WH_DATA.0	 := GVL1.hwo_digitalAlarms[6].0	;	(*	DI:97	WH ALARM MUTE P/B	*)
WH_DATA.1	 := GVL1.hwo_digitalAlarms[6].1	;	(*	DI:98	STGR JOYSTICK CONTROL FAIL ALARM	*)
WH_DATA.2	 := GVL1.hwo_digitalAlarms[6].2	;	(*	DI:99	GEN.ALARM MAIN SUPPLY FAILURE	*)
WH_DATA.3	 := GVL1.hwo_digitalAlarms[6].3	;	(*	DI:100	GEN.ALARM ALT.SUPPLY FAILURE	*)
WH_DATA.4	 := GVL1.hwo_digitalAlarms[6].4	;	(*	DI:101	NAV.LIGHT POWER FAILURE	*)
WH_DATA.5	 := GVL1.hwo_digitalAlarms[6].5	;	(*	DI:102	NAV.LIGHT SYSTEM FAULT	*)
WH_DATA.6	 := GVL1.hwo_digitalAlarms[6].6	;	(*	DI:103	FIRE ALARM SYSTEM FAULT	*)
WH_DATA.7	 := GVL1.hwo_digitalAlarms[6].7	;	(*	DI:104	FIRE ALARM ACTVATED	*)
WH_DATA.8	 := GVL1.hwo_digitalAlarms[6].8	;	(*	DI:105	AUTO PILOT FAIL ALARM	*)
WH_DATA.9	 := GVL1.hwo_digitalAlarms[6].9	;	(*	DI:106	GAS DETECTION SYSTEM POWER FAIL	*)
WH_DATA.10	 := GVL1.hwo_digitalAlarms[6].10	;	(*	DI:107	H2S ALARM ACTIVATED	*)
WH_DATA.11	 := GVL1.hwo_digitalAlarms[6].11	;	(*	DI:108	LEL ALARM ACTIVATED	*)
WH_DATA.12	 := GVL1.hwo_digitalAlarms[6].12	;	(*	DI:109	WH AREA REF. LEAKAGE ALARM 	*)
WH_DATA.13	 := GVL1.hwo_digitalAlarms[6].13	;	(*	DI:110	PASSENGER AREA REF. LEAKAGE ALARM 	*)
WH_DATA.14	 := GVL1.hwo_digitalAlarms[6].14	;	(*	DI:111	DEPTH BELOW KEEL LOWER THAN SET.P 	*)
WH_DATA.15	 := GVL1.hwo_digitalAlarms[6].15	;	(*	DI:112	GMDSS COMMON ALRM	*)
						
MP1_DATA.0	 := GVL1.hwo_digitalAlarms[7].0	;	(*	DI:113	PORT ME COMMON ALARM	*)
MP1_DATA.1	 := GVL1.hwo_digitalAlarms[7].1	;	(*	DI:114	STBD ME COMMON ALARM	*)
MP1_DATA.2	 := GVL1.hwo_digitalAlarms[7].2	;	(*	DI:115	CENTER ME COMMON ALARM	*)
MP1_DATA.3	 := GVL1.hwo_digitalEvents[7].3	;	(*	DI:116	AUX COOLING PUMP-1 RUNNING	*)
MP1_DATA.4	 := GVL1.hwo_digitalAlarms[7].4	;	(*	DI:117	AUX COOLING PUMP-1 TRIP	*)
MP1_DATA.5	 := GVL1.hwo_digitalAlarms[7].5	;	(*	DI:118	FO PURIFIER COMMON ALRM	*)
MP1_DATA.6	 := GVL1.hwo_digitalAlarms[7].6	;	(*	DI:119	MSB: PREF. TRIP ALARM	*)
MP1_DATA.7	 := GVL1.hwo_digitalAlarms[7].7	;	(*	DI:120	MSB: 440V EARTH FAULT ALARM	*)
MP1_DATA.8	 := GVL1.hwo_digitalAlarms[7].8	;	(*	DI:121	MSB: 220V EARTH FAULT ALARM	*)
MP1_DATA.9	 := GVL1.hwo_digitalAlarms[7].9	;	(*	DI:122	MSB: 24VDC SUPPLY FAIL ALARM	*)
MP1_DATA.10	 := GVL1.hwo_digitalAlarms[7].10	;	(*	DI:123	MSB: ABNORMAL ALARM	*)
MP1_DATA.11	 := GVL1.hwo_digitalAlarms[7].11	;	(*	DI:124	AMS AC SUPPLY FAIL	*)
MP1_DATA.12	 := GVL1.hwo_digitalAlarms[7].12	;	(*	DI:125	AMS DC SUPPLY FAIL	*)
MP1_DATA.13	 := GVL1.hwo_digitalAlarms[7].13	;	(*	DI:126	ALRM MUTE AMS PANEL	*)
MP1_DATA.14	 := GVL1.hwo_digitalAlarms[7].14	;	(*	DI:127	BT ENGINE COMMON ALARM	*)
MP1_DATA.15	 := GVL1.hwo_digitalAlarms[7].15	;	(*	DI:128	ACCOM PASSAGE REF. LEAKAGE ALARM	*)
						
MP2_DATA.0	 := GVL1.hwo_digitalAlarms[8].0	;	(*	DI:129	SPARE	*)
MP2_DATA.1	 := GVL1.hwo_digitalAlarms[8].1	;	(*	DI:130	SPARE	*)
MP2_DATA.2	 := GVL1.hwo_digitalAlarms[8].2	;	(*	DI:131	SPARE	*)
MP2_DATA.3	 := GVL1.hwo_digitalAlarms[8].3	;	(*	DI:132	SPARE	*)
MP2_DATA.4	 := GVL1.hwo_digitalAlarms[8].4	;	(*	DI:133	SPARE	*)
MP2_DATA.5	 := GVL1.hwo_digitalAlarms[8].5	;	(*	DI:134	SPARE	*)
MP2_DATA.6	 := GVL1.hwo_digitalAlarms[8].6	;	(*	DI:135	SPARE	*)
MP2_DATA.7	 := GVL1.hwo_digitalAlarms[8].7	;	(*	DI:136	SPARE	*)
MP2_DATA.8	 := GVL1.hwo_digitalAlarms[8].8	;	(*	DI:137	SPARE	*)
MP2_DATA.9	 := GVL1.hwo_digitalAlarms[8].9	;	(*	DI:138	SPARE	*)
MP2_DATA.10	 := GVL1.hwo_digitalAlarms[8].10	;	(*	DI:139	SPARE	*)
MP2_DATA.11	 := GVL1.hwo_digitalAlarms[8].11	;	(*	DI:140	SPARE	*)
MP2_DATA.12	 := GVL1.hwo_digitalAlarms[8].12	;	(*	DI:141	SPARE	*)
MP2_DATA.13	 := GVL1.hwo_digitalAlarms[8].13	;	(*	DI:142	SPARE	*)
MP2_DATA.14	 := GVL1.hwo_digitalAlarms[8].14	;	(*	DI:143	SPARE	*)
MP2_DATA.15	 := GVL1.hwo_digitalAlarms[8].15	;	(*	DI:144	SPARE	*)
						
MP3_DATA.0	 := GVL1.hwo_digitalAlarms[9].0	;	(*	DI:145	SPARE	*)
MP3_DATA.1	 := GVL1.hwo_digitalAlarms[9].1	;	(*	DI:146	SPARE	*)
MP3_DATA.2	 := GVL1.hwo_digitalAlarms[9].2	;	(*	DI:147	SPARE	*)
MP3_DATA.3	 := GVL1.hwo_digitalAlarms[9].3	;	(*	DI:148	SPARE	*)
MP3_DATA.4	 := GVL1.hwo_digitalAlarms[9].4	;	(*	DI:149	SPARE	*)
MP3_DATA.5	 := GVL1.hwo_digitalAlarms[9].5	;	(*	DI:150	SPARE	*)
MP3_DATA.6	 := GVL1.hwo_digitalAlarms[9].6	;	(*	DI:151	SPARE	*)
MP3_DATA.7	 := GVL1.hwo_digitalAlarms[9].7	;	(*	DI:152	SPARE	*)
						
IF NOT GVL1.hwo_digitalAlarms[12].11 THEN						
AI1_DATA	:= REAL_TO_WORD (GVL1.hro_Ch0OutVal[2])	;	(*	AI:01-FRESH WATER TANK 1C	*)
AI2_DATA	:= REAL_TO_WORD (GVL1.hro_Ch1OutVal[2])	;	(*	AI:02-FRESH WATER TANK 2C	*)
AI3_DATA	:= REAL_TO_WORD (GVL1.hro_Ch2OutVal[2])	;	(*	AI:03-BLACK WATER TANK	*)
AI4_DATA	:= REAL_TO_WORD (GVL1.hro_Ch3OutVal[2])	;	(*	AI:04-GREY WATER TANK 	*)
AI5_DATA	:= REAL_TO_WORD (GVL1.hro_Ch4OutVal[2])	;	(*	AI:05-FUEL OIL TANK PORT 1P	*)
AI6_DATA	:= REAL_TO_WORD (GVL1.hro_Ch5OutVal[2])	;	(*	AI:06-FUEL OIL TANK STBD 1S	*)
AI7_DATA	:= REAL_TO_WORD (GVL1.hro_Ch6OutVal[2])	;	(*	AI:07-FUEL OIL TANK PORT 3C	*)
AI8_DATA	:= REAL_TO_WORD (GVL1.hro_Ch7OutVal[2])	;	(*	AI:08-BILGE HOLDING TANK	*)
AI9_DATA	:= REAL_TO_WORD (GVL1.hro_Ch8OutVal[2])	;	(*	AI:09-FODS TANK PORT	*)
AI10_DATA	:= REAL_TO_WORD (GVL1.hro_Ch9OutVal[2])	;	(*	AI:10-FODS TANK STDB	*)
AI11_DATA	:= REAL_TO_WORD (GVL1.hro_Ch10OutVal[2])	;	(*	AI:11-SLOPE TANK 	*)
AI12_DATA	:= REAL_TO_WORD (GVL1.hro_Ch11OutVal[2])	;	(*	AI:12-FUEL OIL TANK PORT 2C	*)
AI13_DATA	:= REAL_TO_WORD (GVL1.hro_Ch12OutVal[2])	;	(*	AI:13-FUEL OIL TANK PORT 4P	*)
AI14_DATA	:= REAL_TO_WORD (GVL1.hro_Ch13OutVal[2])	;	(*	AI:14-FUEL OIL TANK STBD 4S	*)

						
						
ELSE						
AI1_DATA	:= 0 ;					
AI2_DATA	:= 0 ;					
AI3_DATA	:= 0 ;					
AI4_DATA	:= 0 ;					
AI5_DATA	:= 0 ;					
AI6_DATA	:= 0 ;					
AI7_DATA	:= 0 ;					
AI8_DATA	:= 0 ;					
AI9_DATA	:= 0 ;					
AI10_DATA	:= 0 ;					
AI11_DATA	:= 0 ;					
AI12_DATA	:= 0 ;					
AI13_DATA	:= 0 ;					
AI14_DATA	:= 0 ;					
END_IF						
						
COM_DATA.0	 := GVL1.hwo_digitalAlarms[12].0	;(*	JB1 DI MODULE COMMS: FAIL	*)		
COM_DATA.1	 := GVL1.hwo_digitalAlarms[12].1	;(*	JB2 DI MODULE COMMS: FAIL	*)		
COM_DATA.2	 := GVL1.hwo_digitalAlarms[12].2	;(*	JB3 DI MODULE COMMS: FAIL	*)		
COM_DATA.3	 := GVL1.hwo_digitalAlarms[12].3	;(*	JB4 DI MODULE COMMS: FAIL	*)		
COM_DATA.4	 := GVL1.hwo_digitalAlarms[12].4	;(*	JB5 DI MODULE COMMS: FAIL	*)		
COM_DATA.5	 := GVL1.hwo_digitalAlarms[12].5	;(*	JB6 DI MODULE COMMS: FAIL	*)		
COM_DATA.6	 := GVL1.hwo_digitalAlarms[12].6	;(*	WH DI MODULE COMMS: FAIL	*)		
COM_DATA.7	 := GVL1.hwo_digitalAlarms[12].7	;(*	MP DI1 MODULE COMMS: FAIL	*)		
COM_DATA.8	 := GVL1.hwo_digitalAlarms[12].8	;(*	MP DI2 MODULE COMMS: FAIL	*)		
COM_DATA.9	 := GVL1.hwo_digitalAlarms[12].9	;(*	MP DIO MODULE COMMS: FAIL	*)		
COM_DATA.10	 := GVL1.hwo_digitalAlarms[12].10	;(*	MP DO MODULE COMMS: FAIL	*)		
COM_DATA.11	 := GVL1.hwo_digitalAlarms[12].11	;(*	MP AI MODULE COMMS: FAIL	*)		
COM_DATA.12	 := GVL1.hwo_digitalAlarms[12].12	; (*	ECR HMI COMMS: FAIL	*)		
COM_DATA.13	 := GVL1.hwo_digitalAlarms[12].13	; (*	WH HMI COMMS: FAIL	*)		
COM_DATA.14	 := GVL1.hwo_digitalAlarms[12].14	; (*	MESS HMI COMMS: FAIL	*)	
	
TK_AL1.0	:=	 GVL1.hwo_analogAlm[0].0   	OR	GVL1.hwo_analogAlm[0].1 	;	(*	AI:01-FW 1C LOW	*)
TK_AL1.1	:=	 GVL1.hwo_analogAlm[0].2	OR	GVL1.hwo_analogAlm[0].5	;	(*	AI:01-FW 1C HIGH	*)
TK_AL1.2	:=	 GVL1.hwo_analogAlm[0].3	OR	GVL1.hwo_analogAlm[0].4	;	(*	AI:01-FW 1C FAULT	*)
TK_AL1.3	:=	 GVL1.hwo_analogAlm[1].0   	OR	GVL1.hwo_analogAlm[1].1 	;	(*	AI:02-FW 2C LOW	*)
TK_AL1.4	:=	 GVL1.hwo_analogAlm[1].2	OR	GVL1.hwo_analogAlm[1].5	;	(*	AI:02-FW 2C HIGH	*)
TK_AL1.5	:=	 GVL1.hwo_analogAlm[1].3	OR	GVL1.hwo_analogAlm[1].4	;	(*	AI:02-FW 2C FAULT	*)
TK_AL1.6	:=	 GVL1.hwo_analogAlm[2].0   	OR	GVL1.hwo_analogAlm[2].1 	;	(*	AI:03-BW LOW	*)
TK_AL1.7	:=	 GVL1.hwo_analogAlm[2].2	OR	GVL1.hwo_analogAlm[2].5	;	(*	AI:03-BW HIGH	*)
TK_AL1.8	:=	 GVL1.hwo_analogAlm[2].3	OR	GVL1.hwo_analogAlm[2].4	;	(*	AI:03-BW FAULT	*)
TK_AL1.9	:=	 GVL1.hwo_analogAlm[3].0   	OR	GVL1.hwo_analogAlm[3].1 	;	(*	AI:04-GW LOW	*)
TK_AL1.10	:=	 GVL1.hwo_analogAlm[3].2	OR	GVL1.hwo_analogAlm[3].5	;	(*	AI:04-GW HIGH	*)
TK_AL1.11	:=	 GVL1.hwo_analogAlm[3].3	OR	GVL1.hwo_analogAlm[3].4	;	(*	AI:04-GW FAULT	*)
TK_AL1.12	:=	 GVL1.hwo_analogAlm[4].0   	OR	GVL1.hwo_analogAlm[4].1 	;	(*	AI:05-FOT1P LOW	*)
TK_AL1.13	:=	 GVL1.hwo_analogAlm[4].2	OR	GVL1.hwo_analogAlm[4].5	;	(*	AI:05-FOT1P HIGH	*)
TK_AL1.14	:=	 GVL1.hwo_analogAlm[4].3	OR	GVL1.hwo_analogAlm[4].4	;	(*	AI:05-FOT1P FAULT	*)
TK_AL1.15	:=	 GVL1.hwo_analogAlm[5].0   	OR	GVL1.hwo_analogAlm[5].1 	;	(*	AI:06-FOT1S LOW	*)
								
TK_AL2.0	:=	 GVL1.hwo_analogAlm[5].2	OR	GVL1.hwo_analogAlm[5].5	;	(*	AI:06-FOT1S HIGH	*)
TK_AL2.1	:=	 GVL1.hwo_analogAlm[5].3	OR	GVL1.hwo_analogAlm[5].4	;	(*	AI:06-FOT1S FAULT	*)
TK_AL2.2	:=	 GVL1.hwo_analogAlm[6].0   	OR	GVL1.hwo_analogAlm[6].1 	;	(*	AI:07-FOT3C LOW	*)
TK_AL2.3	:=	 GVL1.hwo_analogAlm[6].2	OR	GVL1.hwo_analogAlm[6].5	;	(*	AI:07-FOT3C HIGH	*)
TK_AL2.4	:=	 GVL1.hwo_analogAlm[6].3	OR	GVL1.hwo_analogAlm[6].4	;	(*	AI:07-FOT3C FAULT	*)
TK_AL2.5	:=	 GVL1.hwo_analogAlm[7].0   	OR	GVL1.hwo_analogAlm[7].1 	;	(*	AI:08-BILGE.H LOW	*)
TK_AL2.6	:=	 GVL1.hwo_analogAlm[7].2	OR	GVL1.hwo_analogAlm[7].5	;	(*	AI:08-BILGE.H HIGH	*)
TK_AL2.7	:=	 GVL1.hwo_analogAlm[7].3	OR	GVL1.hwo_analogAlm[7].4	;	(*	AI:08-BILGE.H FAULT	*)
TK_AL2.8	:=	 GVL1.hwo_analogAlm[8].0   	OR	GVL1.hwo_analogAlm[8].1 	;	(*	AI:09-FODS P LOW	*)
TK_AL2.9	:=	 GVL1.hwo_analogAlm[8].2	OR	GVL1.hwo_analogAlm[8].5	;	(*	AI:09-FODS P HIGH	*)
TK_AL2.10	:=	 GVL1.hwo_analogAlm[8].3	OR	GVL1.hwo_analogAlm[8].4	;	(*	AI:09-FODS P FAULT	*)
TK_AL2.11	:=	 GVL1.hwo_analogAlm[9].0   	OR	GVL1.hwo_analogAlm[9].1 	;	(*	AI:10-FODS S LOW	*)
TK_AL2.12	:=	 GVL1.hwo_analogAlm[9].2	OR	GVL1.hwo_analogAlm[9].5	;	(*	AI:10-FODS S HIGH	*)
TK_AL2.13	:=	 GVL1.hwo_analogAlm[9].3	OR	GVL1.hwo_analogAlm[9].4	;	(*	AI:10-FODS S FAULT	*)
TK_AL2.14	:=	 GVL1.hwo_analogAlm[10].0  	OR	GVL1.hwo_analogAlm[10].1 	;	(*	AI:11-SLOPE LOW	*)
TK_AL2.15	:=	 GVL1.hwo_analogAlm[10].2	OR	GVL1.hwo_analogAlm[10].5 	;	(*	AI:11-SLOPE HIGH	*)
								
TK_AL3.0	:=	 GVL1.hwo_analogAlm[10].3	OR	GVL1.hwo_analogAlm[10].4	;	(*	AI:11-SLOPE FAULT	*)
TK_AL3.1	:=	 GVL1.hwo_analogAlm[11].0  	OR	GVL1.hwo_analogAlm[11].1 	;	(*	AI:12-FOT2C LOW	*)
TK_AL3.2	:=	 GVL1.hwo_analogAlm[11].2	OR	GVL1.hwo_analogAlm[11].5	;	(*	AI:12-FOT2C HIGH	*)
TK_AL3.3	:=	 GVL1.hwo_analogAlm[11].3	OR	GVL1.hwo_analogAlm[11].4	;	(*	AI:12-FOT2C FAULT	*)
TK_AL3.4	:=	 GVL1.hwo_analogAlm[12].0 	OR	GVL1.hwo_analogAlm[12].1 	;	(*	AI:13-FOT4P LOW	*)
TK_AL3.5	:=	 GVL1.hwo_analogAlm[12].2	OR	GVL1.hwo_analogAlm[12].5	;	(*	AI:13-FOT4P HIGH	*)
TK_AL3.6	:=	 GVL1.hwo_analogAlm[12].3	OR	GVL1.hwo_analogAlm[12].4	;	(*	AI:13-FOT4P FAULT	*)
TK_AL3.7	:=	 GVL1.hwo_analogAlm[13].0 	OR	GVL1.hwo_analogAlm[13].1 	;	(*	AI:14-FOT4S LOW	*)
TK_AL3.8	:=	 GVL1.hwo_analogAlm[13].2	OR	GVL1.hwo_analogAlm[13].5	;	(*	AI:14-FOT4S HIGH	*)
TK_AL3.9	:=	 GVL1.hwo_analogAlm[13].3	OR	GVL1.hwo_analogAlm[13].4	;	(*	AI:14-FOT4S FAULT	*)
END_ACTION

END_PROGRAM

// Device/Application/fb_alarmEvent
FUNCTION_BLOCK fb_alarmEvent
VAR_INPUT
	wi_input: WORD;
	wi_set: WORD :=65535;
	wai_delay: ARRAY[0..15] OF WORD;
	wi_inhibit: WORD;
	wi_inhibitJm: WORD;
	wi_interlock: WORD;
	wi_alarmEvent: WORD;
	xi_reset: BOOL;
	xi_ack: BOOL;
	
END_VAR
VAR_OUTPUT
	wo_alarm: WORD;
	wo_event: WORD;
	wo_alarmLa : WORD;
	xo_buzzer: BOOL;
	xo_ind: BOOL;
	xo_indLa: BOOL;
	wo_inhTot: WORD;
END_VAR
VAR
	AlarmOutTemp: WORD;
	AlarmDelayTemp: ARRAY[0..15] OF TIME;
	

	HighInterlock1: WORD;
	HighInterlock2: WORD;
	LowInterlock1: WORD;
	LowInterlock2: WORD;
	
	TR1: TON;
	TR2: TON;
	TR3: TON;
	TR4: TON;
	TR5: TON;
	TR6: TON;
	TR7: TON;
	TR8: TON;
	TR9: TON;
	TR10: TON;
	TR11: TON;
	TR12: TON;
	TR13: TON;
	TR14: TON;
	TR15: TON;
	TR16: TON;
	AlarmOut1: TP;
	AlarmOut2: TP;
	AlarmOut3: TP;
	AlarmOut4: TP;
	AlarmOut5: TP;
	AlarmOut6: TP;
	AlarmOut7: TP;
	AlarmOut8: TP;
	AlarmOut9: TP;
	AlarmOut10: TP;
	AlarmOut11: TP;
	AlarmOut12: TP;
	AlarmOut13: TP;
	AlarmOut14: TP;
	AlarmOut15: TP;
	AlarmOut16: TP;
	x_reset1: BOOL;
	x_reset2: BOOL;
	x_reset3: BOOL;
	x_reset4: BOOL;
	x_reset5: BOOL;
	x_reset6: BOOL;
	x_reset7: BOOL;
	x_reset8: BOOL;
	x_reset9: BOOL;
	x_reset10: BOOL;
	x_reset11: BOOL;
	x_reset12: BOOL;
	x_reset13: BOOL;
	x_reset14: BOOL;
	x_reset15: BOOL;
	x_reset16: BOOL;
END_VAR

(*Alarm1*)

(*x_reset*)
IF wo_alarm.0 AND xi_reset THEN
x_reset1:= TRUE;
ELSE
x_reset1:= FALSE;
END_IF


(*Time delay*)
TR1(IN:= , PT:= , Q=> , ET=> );
TR1.IN:=AlarmOutTemp.0;
TR1.PT:= AlarmDelayTemp[0];
AlarmDelayTemp[0]:=WORD_TO_TIME ( wai_delay[0]*1000);

(*Alarm condition:- Set NO/NC, Inhibit, x_reset*)
IF ((wi_input.0=1 AND wi_set.0=1) OR (wi_input.0=0 AND wi_set.0=0)) AND wi_inhibit.0=0 AND wi_inhibitJm.0=0 AND x_reset1=0
THEN
AlarmOutTemp.0:=1;
ELSE
AlarmOutTemp.0:=0;
END_IF


(*Final alarm and event output with delay*)
wo_alarm.0:=TR1.Q AND wi_alarmEvent.0 AND NOT wi_interlock.0;
wo_event.0:=TR1.Q ;
(*Final alarm single pulse latched till acknowledge*)
AlarmOut1(IN:=wo_alarm.0 , PT:= T#1s, Q=> , ET=> );
IF (AlarmOut1.Q OR wo_alarmLa.0) AND NOT xi_ack THEN wo_alarmLa.0:=1; ELSE wo_alarmLa.0:=0; END_IF
(*------------------------------------------------------------------------------------------------------------------------------*)

(*Alarm2*)

(*x_reset*)
IF wo_alarm.1 AND xi_reset THEN
x_reset2:= TRUE;
ELSE
x_reset2:= FALSE;
END_IF


(*Time delay*)
TR2(IN:= , PT:= , Q=> , ET=> );
TR2.IN:=AlarmOutTemp.1;
TR2.PT:= AlarmDelayTemp[1];
AlarmDelayTemp[1]:=WORD_TO_TIME ( wai_delay[1]*1000);

(*Alarm condition:- Set NO/NC, Inhibit, x_reset*)
IF ((wi_input.1=1 AND wi_set.1=1) OR (wi_input.1=0 AND wi_set.1=0)) AND wi_inhibit.1=0 AND wi_inhibitJm.1=0  AND x_reset2=0
THEN
AlarmOutTemp.1:=1;
ELSE
AlarmOutTemp.1:=0;
END_IF


(*Final alarm and event output with delay*)
wo_alarm.1:=TR2.Q AND wi_alarmEvent.1 AND NOT wi_interlock.1;
wo_event.1:=TR2.Q;
(*Final alarm single pulse latched till acknowledge*)
AlarmOut2(IN:=wo_alarm.1 , PT:= T#1s, Q=> , ET=> );
IF (AlarmOut2.Q OR wo_alarmLa.1) AND NOT xi_ack THEN wo_alarmLa.1:=1; ELSE wo_alarmLa.1:=0; END_IF

(*------------------------------------------------------------------------------------------------------------------------------*)

(*Alarm3*)

(*x_reset*)
IF wo_alarm.2 AND xi_reset THEN
x_reset3:= TRUE;
ELSE
x_reset3:= FALSE;
END_IF


(*Time delay*)
TR3(IN:= , PT:= , Q=> , ET=> );
TR3.IN:=AlarmOutTemp.2;
TR3.PT:= AlarmDelayTemp[2];
AlarmDelayTemp[2]:=WORD_TO_TIME ( wai_delay[2]*1000);

(*Alarm condition:- Set NO/NC, Inhibit, x_reset*)
IF ((wi_input.2=1 AND wi_set.2=1) OR (wi_input.2=0 AND wi_set.2=0)) AND wi_inhibit.2=0 AND wi_inhibitJm.2=0   AND x_reset3=0
THEN
AlarmOutTemp.2:=1;
ELSE
AlarmOutTemp.2:=0;
END_IF

(*Final alarm and event output with delay*)
wo_alarm.2:=TR3.Q AND wi_alarmEvent.2 AND NOT wi_interlock.2;
wo_event.2:=TR3.Q;
(*Final alarm single pulse latched till acknowledge*)
AlarmOut3(IN:=wo_alarm.2 , PT:= T#1s, Q=> , ET=> );
IF (AlarmOut3.Q OR wo_alarmLa.2) AND NOT xi_ack THEN wo_alarmLa.2:=1; ELSE wo_alarmLa.2:=0; END_IF
(*------------------------------------------------------------------------------------------------------------------------------*)

(*Alarm4*)

(*x_reset*)
IF wo_alarm.3 AND xi_reset THEN
x_reset4:= TRUE;
ELSE
x_reset4:= FALSE;
END_IF


(*Time delay*)
TR4(IN:= , PT:= , Q=> , ET=> );
TR4.IN:=AlarmOutTemp.3;
TR4.PT:= AlarmDelayTemp[3];
AlarmDelayTemp[3]:=WORD_TO_TIME ( wai_delay[3]*1000);

(*Alarm condition:- Set NO/NC, Inhibit, x_reset*)
IF ((wi_input.3=1 AND wi_set.3=1) OR (wi_input.3=0 AND wi_set.3=0)) AND wi_inhibit.3=0 AND wi_inhibitJm.3=0  AND x_reset4=0
THEN
AlarmOutTemp.3:=1;
ELSE
AlarmOutTemp.3:=0;
END_IF

(*Final alarm and event output with delay*)
wo_alarm.3:=TR4.Q AND wi_alarmEvent.3 AND NOT wi_interlock.3;
wo_event.3:=TR4.Q;
(*Final alarm single pulse latched till acknowledge*)
AlarmOut4(IN:=wo_alarm.3 , PT:= T#1s, Q=> , ET=> );
IF (AlarmOut4.Q OR wo_alarmLa.3) AND NOT xi_ack THEN wo_alarmLa.3:=1; ELSE wo_alarmLa.3:=0; END_IF
(*------------------------------------------------------------------------------------------------------------------------------*)

(*Alarm5*)

(*x_reset*)
IF wo_alarm.4 AND xi_reset THEN
x_reset5:= TRUE;
ELSE
x_reset5:= FALSE;
END_IF


(*Time delay*)
TR5(IN:= , PT:= , Q=> , ET=> );
TR5.IN:=AlarmOutTemp.4;
TR5.PT:= AlarmDelayTemp[4];
AlarmDelayTemp[4]:=WORD_TO_TIME ( wai_delay[4]*1000);

(*Alarm condition:- Set NO/NC, Inhibit, x_reset*)
IF ((wi_input.4=1 AND wi_set.4=1) OR (wi_input.4=0 AND wi_set.4=0)) AND wi_inhibit.4=0 AND wi_inhibitJm.4=0   AND x_reset5=0
THEN
AlarmOutTemp.4:=1;
ELSE
AlarmOutTemp.4:=0;
END_IF

(*Final alarm and event output with delay*)
wo_alarm.4:=TR5.Q AND wi_alarmEvent.4 AND NOT wi_interlock.4;
wo_event.4:=TR5.Q;
(*Final alarm single pulse latched till acknowledge*)
AlarmOut5(IN:=wo_alarm.4 , PT:= T#1s, Q=> , ET=> );
IF (AlarmOut5.Q OR wo_alarmLa.4) AND NOT xi_ack THEN wo_alarmLa.4:=1; ELSE wo_alarmLa.4:=0; END_IF

(*------------------------------------------------------------------------------------------------------------------------------*)

(*Alarm6*)

(*x_reset*)
IF wo_alarm.5 AND xi_reset THEN
x_reset6:= TRUE;
ELSE
x_reset6:= FALSE;
END_IF


(*Time delay*)
TR6(IN:= , PT:= , Q=> , ET=> );
TR6.IN:=AlarmOutTemp.5;
TR6.PT:= AlarmDelayTemp[5];
AlarmDelayTemp[5]:=WORD_TO_TIME ( wai_delay[5]*1000);

(*Alarm condition:- Set NO/NC, Inhibit, x_reset*)
IF ((wi_input.5=1 AND wi_set.5=1) OR (wi_input.5=0 AND wi_set.5=0)) AND wi_inhibit.5=0 AND wi_inhibitJm.5=0   AND x_reset6=0
THEN
AlarmOutTemp.5:=1;
ELSE
AlarmOutTemp.5:=0;
END_IF

(*Final alarm and event output with delay*)
wo_alarm.5:=TR6.Q AND wi_alarmEvent.5 AND NOT wi_interlock.5;
wo_event.5:=TR6.Q;
(*Final alarm single pulse latched till acknowledge*)
AlarmOut6(IN:=wo_alarm.5 , PT:= T#1s, Q=> , ET=> );
IF (AlarmOut6.Q OR wo_alarmLa.5) AND NOT xi_ack THEN wo_alarmLa.5:=1; ELSE wo_alarmLa.5:=0; END_IF
(*------------------------------------------------------------------------------------------------------------------------------*)

(*Alarm7*)

(*x_reset*)
IF wo_alarm.6 AND xi_reset THEN
x_reset7:= TRUE;
ELSE
x_reset7:= FALSE;
END_IF


(*Time delay*)
TR7(IN:= , PT:= , Q=> , ET=> );
TR7.IN:=AlarmOutTemp.6;
TR7.PT:= AlarmDelayTemp[6];
AlarmDelayTemp[6]:=WORD_TO_TIME ( wai_delay[6]*1000);

(*Alarm condition:- Set NO/NC, Inhibit, x_reset*)
IF ((wi_input.6=1 AND wi_set.6=1) OR (wi_input.6=0 AND wi_set.6=0)) AND wi_inhibit.6=0 AND wi_inhibitJm.6=0   AND x_reset7=0
THEN
AlarmOutTemp.6:=1;
ELSE
AlarmOutTemp.6:=0;
END_IF


(*Final alarm and event output with delay*)
wo_alarm.6:=TR7.Q AND wi_alarmEvent.6 AND NOT wi_interlock.6;
wo_event.6:=TR7.Q;
(*Final alarm single pulse latched till acknowledge*)
AlarmOut7(IN:=wo_alarm.6 , PT:= T#1s, Q=> , ET=> );
IF (AlarmOut7.Q OR wo_alarmLa.6) AND NOT xi_ack THEN wo_alarmLa.6:=1; ELSE wo_alarmLa.6:=0; END_IF
(*------------------------------------------------------------------------------------------------------------------------------*)

(*Alarm8*)

(*x_reset*)
IF wo_alarm.7 AND xi_reset THEN
x_reset8:= TRUE;
ELSE
x_reset8:= FALSE;
END_IF


(*Time delay*)
TR8(IN:= , PT:= , Q=> , ET=> );
TR8.IN:=AlarmOutTemp.7;
TR8.PT:= AlarmDelayTemp[7];
AlarmDelayTemp[7]:=WORD_TO_TIME ( wai_delay[7]*1000);

(*Alarm condition:- Set NO/NC, Inhibit, x_reset*)
IF ((wi_input.7=1 AND wi_set.7=1) OR (wi_input.7=0 AND wi_set.7=0)) AND wi_inhibit.7=0 AND wi_inhibitJm.7=0   AND x_reset8=0
THEN
AlarmOutTemp.7:=1;
ELSE
AlarmOutTemp.7:=0;
END_IF

(*Final alarm and event output with delay*)
wo_alarm.7:=TR8.Q AND wi_alarmEvent.7 AND NOT wi_interlock.7;
wo_event.7:=TR8.Q;
(*Final alarm single pulse latched till acknowledge*)
AlarmOut8(IN:=wo_alarm.7 , PT:= T#1s, Q=> , ET=> );
IF (AlarmOut8.Q OR wo_alarmLa.7) AND NOT xi_ack THEN wo_alarmLa.7:=1; ELSE wo_alarmLa.7:=0; END_IF
(*------------------------------------------------------------------------------------------------------------------------------*)

(*Alarm9*)

(*x_reset*)
IF wo_alarm.8 AND xi_reset THEN
x_reset9:= TRUE;
ELSE
x_reset9:= FALSE;
END_IF


(*Time delay*)
TR9(IN:= , PT:= , Q=> , ET=> );
TR9.IN:=AlarmOutTemp.8;
TR9.PT:= AlarmDelayTemp[8];
AlarmDelayTemp[8]:=WORD_TO_TIME ( wai_delay[8]*1000);

(*Alarm condition:- Set NO/NC, Inhibit, x_reset*)
IF ((wi_input.8=1 AND wi_set.8=1) OR (wi_input.8=0 AND wi_set.8=0)) AND wi_inhibit.8=0 AND wi_inhibitJm.8=0   AND x_reset9=0
THEN
AlarmOutTemp.8:=1;
ELSE
AlarmOutTemp.8:=0;
END_IF

(*Final alarm and event output with delay*)
wo_alarm.8:=TR9.Q AND wi_alarmEvent.8 AND NOT wi_interlock.8;
wo_event.8:=TR9.Q;
(*Final alarm single pulse latched till acknowledge*)
AlarmOut9(IN:=wo_alarm.8 , PT:= T#1s, Q=> , ET=> );
IF (AlarmOut9.Q OR wo_alarmLa.8) AND NOT xi_ack THEN wo_alarmLa.8:=1; ELSE wo_alarmLa.8:=0; END_IF
(*------------------------------------------------------------------------------------------------------------------------------*)

(*Alarm10*)

(*x_reset*)
IF wo_alarm.9 AND xi_reset THEN
x_reset10:= TRUE;
ELSE
x_reset10:= FALSE;
END_IF


(*Time delay*)
TR10(IN:= , PT:= , Q=> , ET=> );
TR10.IN:=AlarmOutTemp.9;
TR10.PT:= AlarmDelayTemp[9];
AlarmDelayTemp[9]:=WORD_TO_TIME ( wai_delay[9]*1000);

(*Alarm condition:- Set NO/NC, Inhibit, x_reset*)
IF ((wi_input.9=1 AND wi_set.9=1) OR (wi_input.9=0 AND wi_set.9=0)) AND wi_inhibit.9=0 AND wi_inhibitJm.9=0  AND x_reset10=0
THEN
AlarmOutTemp.9:=1;
ELSE
AlarmOutTemp.9:=0;
END_IF

(*Final alarm and event output with delay*)
wo_alarm.9:=TR10.Q AND wi_alarmEvent.9 AND NOT wi_interlock.9;
wo_event.9:=TR10.Q;
(*Final alarm single pulse latched till acknowledge*)
AlarmOut10(IN:=wo_alarm.9 , PT:= T#1s, Q=> , ET=> );
IF (AlarmOut10.Q OR wo_alarmLa.9) AND NOT xi_ack THEN wo_alarmLa.9:=1; ELSE wo_alarmLa.9:=0; END_IF
(*------------------------------------------------------------------------------------------------------------------------------*)

(*Alarm11*)

(*x_reset*)
IF wo_alarm.10 AND xi_reset THEN
x_reset11:= TRUE;
ELSE
x_reset11:= FALSE;
END_IF


(*Time delay*)
TR11(IN:= , PT:= , Q=> , ET=> );
TR11.IN:=AlarmOutTemp.10;
TR11.PT:= AlarmDelayTemp[10];
AlarmDelayTemp[10]:=WORD_TO_TIME ( wai_delay[10]*1000);

(*Alarm condition:- Set NO/NC, Inhibit, x_reset*)
IF ((wi_input.10=1 AND wi_set.10=1) OR (wi_input.10=0 AND wi_set.10=0)) AND wi_inhibit.10=0 AND wi_inhibitJm.10=0   AND x_reset11=0
THEN
AlarmOutTemp.10:=1;
ELSE
AlarmOutTemp.10:=0;
END_IF

(*Final alarm and event output with delay*)
wo_alarm.10:=TR11.Q AND wi_alarmEvent.10 AND NOT wi_interlock.10;
wo_event.10:=TR11.Q;
(*Final alarm single pulse latched till acknowledge*)
AlarmOut11(IN:=wo_alarm.10 , PT:= T#1s, Q=> , ET=> );
IF (AlarmOut11.Q OR wo_alarmLa.10) AND NOT xi_ack THEN wo_alarmLa.10:=1; ELSE wo_alarmLa.10:=0; END_IF
(*------------------------------------------------------------------------------------------------------------------------------*)

(*Alarm12*)

(*x_reset*)
IF wo_alarm.11 AND xi_reset THEN
x_reset12:= TRUE;
ELSE
x_reset12:= FALSE;
END_IF


(*Time delay*)
TR12(IN:= , PT:= , Q=> , ET=> );
TR12.IN:=AlarmOutTemp.11;
TR12.PT:= AlarmDelayTemp[11];
AlarmDelayTemp[11]:=WORD_TO_TIME ( wai_delay[11]*1000);

(*Alarm condition:- Set NO/NC, Inhibit, x_reset*)
IF ((wi_input.11=1 AND wi_set.11=1) OR (wi_input.11=0 AND wi_set.11=0)) AND wi_inhibit.11=0 AND wi_inhibitJm.11=0   AND x_reset12=0
THEN
AlarmOutTemp.11:=1;
ELSE
AlarmOutTemp.11:=0;
END_IF

(*Final alarm and event output with delay*)
wo_alarm.11:=TR12.Q AND wi_alarmEvent.11 AND NOT wi_interlock.11;
wo_event.11:=TR12.Q;
(*Final alarm single pulse latched till acknowledge*)
AlarmOut12(IN:=wo_alarm.11 , PT:= T#1s, Q=> , ET=> );
IF (AlarmOut12.Q OR wo_alarmLa.11) AND NOT xi_ack THEN wo_alarmLa.11:=1; ELSE wo_alarmLa.11:=0; END_IF

(*------------------------------------------------------------------------------------------------------------------------------*)

(*Alarm13*)

(*x_reset*)
IF wo_alarm.12 AND xi_reset THEN
x_reset13:= TRUE;
ELSE
x_reset13:= FALSE;
END_IF


(*Time delay*)
TR13(IN:= , PT:= , Q=> , ET=> );
TR13.IN:=AlarmOutTemp.12;
TR13.PT:= AlarmDelayTemp[12];
AlarmDelayTemp[12]:=WORD_TO_TIME ( wai_delay[12]*1000);

(*Alarm condition:- Set NO/NC, Inhibit, x_reset*)
IF ((wi_input.12=1 AND wi_set.12=1) OR (wi_input.12=0 AND wi_set.12=0)) AND wi_inhibit.12=0 AND wi_inhibitJm.12=0   AND x_reset13=0
THEN
AlarmOutTemp.12:=1;
ELSE
AlarmOutTemp.12:=0;
END_IF

(*Final alarm and event output with delay*)
wo_alarm.12:=TR13.Q AND wi_alarmEvent.12 AND NOT wi_interlock.12;
wo_event.12:=TR13.Q;
(*Final alarm single pulse latched till acknowledge*)
AlarmOut13(IN:=wo_alarm.12 , PT:= T#1s, Q=> , ET=> );
IF (AlarmOut13.Q OR wo_alarmLa.12) AND NOT xi_ack THEN wo_alarmLa.12:=1; ELSE wo_alarmLa.12:=0; END_IF
(*------------------------------------------------------------------------------------------------------------------------------*)

(*Alarm14*)

(*x_reset*)
IF wo_alarm.13 AND xi_reset THEN
x_reset14:= TRUE;
ELSE
x_reset14:= FALSE;
END_IF


(*Time delay*)
TR14(IN:= , PT:= , Q=> , ET=> );
TR14.IN:=AlarmOutTemp.13;
TR14.PT:= AlarmDelayTemp[13];
AlarmDelayTemp[13]:=WORD_TO_TIME ( wai_delay[13]*1000);

(*Alarm condition:- Set NO/NC, Inhibit, x_reset*)
IF ((wi_input.13=1 AND wi_set.13=1) OR (wi_input.13=0 AND wi_set.13=0)) AND wi_inhibit.13=0 AND wi_inhibitJm.13=0   AND x_reset14=0
THEN
AlarmOutTemp.13:=1;
ELSE
AlarmOutTemp.13:=0;
END_IF

(*Final alarm and event output with delay*)
wo_alarm.13:=TR14.Q AND wi_alarmEvent.13 AND NOT wi_interlock.13;
wo_event.13:=TR14.Q;
(*Final alarm single pulse latched till acknowledge*)
AlarmOut14(IN:=wo_alarm.13 , PT:= T#1s, Q=> , ET=> );
IF (AlarmOut14.Q OR wo_alarmLa.13) AND NOT xi_ack THEN wo_alarmLa.13:=1; ELSE wo_alarmLa.13:=0; END_IF
(*------------------------------------------------------------------------------------------------------------------------------*)

(*Alarm15*)

(*x_reset*)
IF wo_alarm.14 AND xi_reset THEN
x_reset15:= TRUE;
ELSE
x_reset15:= FALSE;
END_IF


(*Time delay*)
TR15(IN:= , PT:= , Q=> , ET=> );
TR15.IN:=AlarmOutTemp.14;
TR15.PT:= AlarmDelayTemp[14];
AlarmDelayTemp[14]:=WORD_TO_TIME ( wai_delay[14]*1000);

(*Alarm condition:- Set NO/NC, Inhibit, x_reset*)
IF ((wi_input.14=1 AND wi_set.14=1) OR (wi_input.14=0 AND wi_set.14=0)) AND wi_inhibit.14=0 AND wi_inhibitJm.14=0  AND x_reset15=0
THEN
AlarmOutTemp.14:=1;
ELSE
AlarmOutTemp.14:=0;
END_IF


(*Final alarm and event output with delay*)
wo_alarm.14:=TR15.Q AND wi_alarmEvent.14 AND NOT wi_interlock.14;
wo_event.14:=TR15.Q;
(*Final alarm single pulse latched till acknowledge*)
AlarmOut15(IN:=wo_alarm.14 , PT:= T#1s, Q=> , ET=> );
IF(AlarmOut15.Q OR wo_alarmLa.14) AND NOT xi_ack THEN wo_alarmLa.14:=1; ELSE wo_alarmLa.14:=0; END_IF
(*------------------------------------------------------------------------------------------------------------------------------*)

(*Alarm16*)

(*x_reset*)
IF wo_alarm.15 AND xi_reset THEN
x_reset16:= TRUE;
ELSE
x_reset16:= FALSE;
END_IF


(*Time delay*)
TR16(IN:= , PT:= , Q=> , ET=> );
TR16.IN:=AlarmOutTemp.15;
TR16.PT:= AlarmDelayTemp[15];
AlarmDelayTemp[15]:=WORD_TO_TIME ( wai_delay[15]*1000);

(*Alarm condition:- Set NO/NC, Inhibit, x_reset*)
IF ((wi_input.15=1 AND wi_set.15=1) OR (wi_input.15=0 AND wi_set.15=0)) AND wi_inhibit.15=0 AND wi_inhibitJm.15=0  AND x_reset16=0
THEN
AlarmOutTemp.15:=1;
ELSE
AlarmOutTemp.15:=0;
END_IF


(*Final alarm and event output with delay*)
wo_alarm.15:=TR16.Q AND wi_alarmEvent.15 AND NOT wi_interlock.15;
wo_event.15:=TR16.Q;
(*Final alarm single pulse latched till acknowledge*)
AlarmOut16(IN:=wo_alarm.15 , PT:= T#1s, Q=> , ET=> );
IF (AlarmOut16.Q OR wo_alarmLa.15) AND NOT xi_ack THEN wo_alarmLa.15:=1; ELSE wo_alarmLa.15:=0; END_IF

(*common buzzer out*)

IF AlarmOut1.Q OR AlarmOut2.Q OR AlarmOut3.Q OR AlarmOut4.Q OR AlarmOut5.Q OR AlarmOut6.Q OR AlarmOut7.Q OR AlarmOut8.Q
OR AlarmOut9.Q OR AlarmOut10.Q OR AlarmOut11.Q OR AlarmOut12.Q OR AlarmOut13.Q OR AlarmOut14.Q OR AlarmOut15.Q OR AlarmOut16.Q THEN
xo_buzzer := 1;
ELSE
xo_buzzer := 0;
END_IF
(*common indication out*)
IF wo_alarm.0 OR wo_alarm.1 OR wo_alarm.2 OR wo_alarm.3 OR wo_alarm.4 OR wo_alarm.5 OR wo_alarm.6
OR wo_alarm.7 OR wo_alarm.8 OR wo_alarm.9 OR wo_alarm.10 OR wo_alarm.11 OR wo_alarm.12 OR wo_alarm.13
OR wo_alarm.14 OR wo_alarm.15 THEN
xo_ind := 1;
ELSE
xo_ind := 0;
END_IF
(*common indication out single pulse latched till acknowledge*)
IF wo_alarmLa.0 OR wo_alarmLa.1 OR wo_alarmLa.2 OR wo_alarmLa.3 OR wo_alarmLa.4 OR wo_alarmLa.5 OR wo_alarmLa.6
OR wo_alarmLa.7 OR wo_alarmLa.8 OR wo_alarmLa.9 OR wo_alarmLa.10 OR wo_alarmLa.11 OR wo_alarmLa.12 OR wo_alarmLa.13
OR wo_alarmLa.14 OR wo_alarmLa.15 THEN
xo_indLa := 1;
ELSE
xo_indLa := 0;
END_IF

(*Total inhibited alarms from Jmobile*)
wo_inhTot := BOOL_TO_WORD(wi_inhibitJm.0) + BOOL_TO_WORD(wi_inhibitJm.1) + BOOL_TO_WORD(wi_inhibitJm.2)
 + BOOL_TO_WORD(wi_inhibitJm.3) + BOOL_TO_WORD(wi_inhibitJm.4) + BOOL_TO_WORD(wi_inhibitJm.5) + BOOL_TO_WORD(wi_inhibitJm.6)
 + BOOL_TO_WORD(wi_inhibitJm.7) + BOOL_TO_WORD(wi_inhibitJm.8) + BOOL_TO_WORD(wi_inhibitJm.9) + BOOL_TO_WORD(wi_inhibitJm.10)
 + BOOL_TO_WORD(wi_inhibitJm.11) + BOOL_TO_WORD(wi_inhibitJm.12) + BOOL_TO_WORD(wi_inhibitJm.13) + BOOL_TO_WORD(wi_inhibitJm.14)
 + BOOL_TO_WORD(wi_inhibitJm.15);

END_FUNCTION_BLOCK

// Device/Application/fb_tankMonitor
FUNCTION_BLOCK fb_tankMonitor
VAR_INPUT
	wi_sensorVal	: WORD;
	wi_samplingIn	: ARRAY[0..20] OF  WORD;
	wi_samplingOut	: ARRAY[0..20] OF  WORD;

	wi_chPara	: WORD;(*0:inhL1, 1:inhL2, 2:inhL3, 3:inhCable break, 4:inhOver range, 5:buz en L1, 6:buz en L2, 7:buz en L3, 8:buz en err1, 9:buz en err2, 10:inhL4, 11:buz en L4, 12: Auto filter enable
							13:Fill input sensor min value and range when tank empty, 14: Fill input sensor max value and range when tank full*)
	wi_chParaJm	: WORD;	
	xi_comErr	:BOOL;
	xi_ack	:BOOL;
END_VAR
VAR_OUTPUT
	ro_pressOut	:REAL;
	ro_htOut	:REAL;
	ro_volOut	:REAL;
	ro_perOut	:REAL;
	ro_curOut	:REAL;
	wo_alarmOut	 : WORD;(*alarm out steady*)
	wo_alarmOutp	 : WORD;(*alarm out single pulse latched till acknowledge*)
	xo_buzPulse	: BOOL;
	xo_ind	:BOOL;
	wo_alarmMsg	:WORD;(*Alarm msg*)
	wo_inhTot :WORD;
END_VAR
VAR
	r_sensorValtemp0 : REAL;
	r_sensorValtemp1 : REAL;
	r_sensorValtemp2 : REAL;
	r_sensorValtemp3 : REAL;
	r_sensorVal	: REAL;
	r_sensorValtemp	:REAL;
	w_alarmOutp_temp	 : WORD;
	ton_delay1	:TON;
	ton_delay2	:TON;
	ton_delay3	:TON;
	ton_delay4	:TON;
	ton_delay5	:TON;
	ton_delay6	:TON;
	tp_almPulse1	:TP;
	tp_almPulse2	:TP;
	tp_almPulse3	:TP;
	tp_almPulse4	:TP;
	tp_almPulse5	:TP;
	tp_almPulse6	:TP;
	x_alarm1Temp1	:BOOL;
	x_alarm2Temp1	:BOOL;
	x_alarm3Temp1	:BOOL;
	x_alarm4Temp1	:BOOL;
	x_alarm5Temp1	:BOOL;
	x_alarm6Temp1	:BOOL;
	LinScale1: fb_linScaleR;
	LinScale2: fb_linScaleR;
	r_valOut: REAL;
	r_pressOut: REAL;
	NonLinScale1: fb_nonLinScale20;
	r_volOut	:REAL;
	r_volOut1	:REAL;
	r_htOut	:REAL;
	r_htOut1	:REAL;
	linScale_r0: fb_linScaleR;
	filter_SH2: sh_2;
	fluctDet1: fb_fluctDet;
END_VAR
VAR_IN_OUT
	ri_chSP	: ARRAY[0..23] OF REAL;(*0:L1Lt, 1:L2Lt, 2:L3Lt, 3:L1delay, 4:L2delay, 5:L3delay,6:Errdelay,
											7:ErrFactor, 8:SensorValMin,9:SensorValMax, 10:SensorRangeMin, 11:SensorRangeMax, 12:filterVal, 
											13:L4Lt, 14:L4delay, 15:heightMin, 16:heightMax, 17:density, 18:unusable , 19:height offset in mm, 
											Auto filter-->20: rate of change, 21: sampling time, 22:sample hold time, 23:filter time constant*)
END_VAR

(*fluctDet1(ri_in:=wi_sensorVal , wi_setVal:=1020 , xo_valFluct=> );*)
fluctDet1(
	ri_in:=wi_sensorVal ,
	ri_rocVal:= ri_chSP[20],
	ri_sampTime:= ri_chSP[21],
	ri_sholdT:=ri_chSP[22] ,
	xo_valFluct=> );
IF fluctDet1.xo_valFluct AND wi_chPara.12 THEN filter_SH2.PT := REAL_TO_TIME ( ri_chSP[23]*1000); ELSE filter_SH2.PT :=REAL_TO_TIME ( ri_chSP[12]*1000); END_IF
filter_SH2(
	in:=wi_sensorVal ,
	PT:= ,
	N:= 16,
	disc:=0 ,
	out=> r_sensorValtemp1,
	trig=> ,
	avg=> r_sensorValtemp0,
	high=> ,
	low=> );
IF (fluctDet1.xo_valFluct AND wi_chPara.12) OR (ri_chSP[12] > 0) THEN r_sensorValtemp2:= r_sensorValtemp0; ELSE r_sensorValtemp2:= r_sensorValtemp1; END_IF

IF  r_sensorValtemp1 = 3 THEN r_sensorValtemp3 := 0; ELSE r_sensorValtemp3 :=  r_sensorValtemp2; END_IF(*return to 0 incase of cable break*)
ro_curOut :=  (20 * r_sensorValtemp3)/4095;(*-->convert  A/D row value to mA-->for 0-20mA input-->	ro_curOut := (20 - 0) / (32760 - 0) * (r_sensorValtemp3 - 0) + 0;*)
(*-->convert  A/D row value to mA-->for 4-20mA input-->	ro_curOut := (20 - 4) / (32760 - 0) * (r_sensorValtemp3 - 0) + 4;*)
r_sensorValtemp := ro_curOut* ri_chSP[7]; (*eror compensation*)
(*method 2 calibration*)

IF wi_chPara.13 THEN ri_chSP[8]:=r_sensorValtemp; ri_chSP[10]:=(ri_chSP[15] * ri_chSP[17] * 9.8066)/1000; END_IF(*Tank empty set*)
IF wi_chPara.14 THEN ri_chSP[9]:=r_sensorValtemp; ri_chSP[11]:=(ri_chSP[16] * ri_chSP[17] * 9.8066)/1000; END_IF(*Tank full set*)
(*scale to output value as per output range given*)
LinScale1(
	input:= r_sensorValtemp,
	xmax:= ri_chSP[9],
	xmin:= ri_chSP[8],
	ymax:= ri_chSP[11],
	ymin:= ri_chSP[10],
	result=> r_pressOut,
	error=> );
ro_pressOut:=r_pressOut ;

(*Liquid height = Pressure / ( Liquid density * Gravity)          -> Pressure in pascal*)
IF ri_chSP[17] > 0 THEN
r_htOut1 := (ro_pressOut * 1000) / (ri_chSP[17] *9.8066);(*height in mm*)
ELSE r_htOut1 :=0; END_IF

IF r_htOut1 > 10 AND ri_chSP[19] > 0 THEN r_htOut := r_htOut1 + ri_chSP[19];(*Added height +offset in mm*)
ELSE IF r_htOut1 >= -ri_chSP[19] AND ri_chSP[19] < 0 THEN r_htOut := r_htOut1 + ri_chSP[19];(*Added height -offset in mm*)
ELSE IF r_htOut1 < -ri_chSP[19] AND ri_chSP[19] < 0 THEN r_htOut := 0;(*Added height -offset in mm*)
ELSE r_htOut := r_htOut1; END_IF END_IF END_IF
IF r_htOut > ri_chSP[16] THEN ro_htOut:=ri_chSP[16];(*Limited to max height*)
ELSE ro_htOut:=r_htOut ; END_IF
(*scale to percentage of height *)
LinScale2(
	input:= ro_htOut,
	xmax:= ri_chSP[16],
	xmin:= ri_chSP[15],
	ymax:= 100,
	ymin:= 0,
	result=> ro_perOut,
	error=> );
(*scale as per sounding table*)
NonLinScale1(
	input:=ro_htOut ,
	xval:=wi_samplingIn ,
	yval:= wi_samplingOut,
	result=>r_volOut ,
	error=> );
IF r_volOut <= ri_chSP[18] AND  ri_chSP[18] > 0  THEN r_volOut1 := 0;
ELSE r_volOut1 :=  r_volOut - ri_chSP[18]; END_IF
ro_volOut	:= r_volOut1;
(*Alarms : level1, level2, ;evel3, cable break, over range, level4*)
IF ro_perOut < ri_chSP[0]AND NOT(wo_alarmOut.3 OR wo_alarmOut.4) THEN x_alarm1Temp1 := 1; ELSE x_alarm1Temp1 := 0; END_IF
ton_delay1(IN:= x_alarm1Temp1 AND NOT wi_chPara.0 AND NOT wi_chParaJm.0, PT:= REAL_TO_TIME ( ri_chSP[3]*1000), Q=> wo_alarmOut.0, ET=> );(*Level 1 alarm steady*)
tp_almPulse1(IN:=wo_alarmOut.0 , PT:= T#1s, Q=> w_alarmOutp_temp.0, ET=> );(*Level 1 alarm single pulse*)
IF (w_alarmOutp_temp.0 OR wo_alarmOutp.0) AND NOT xi_ack THEN wo_alarmOutp.0:=1; ELSE wo_alarmOutp.0:=0; END_IF(*Level 1 alarm single pulse latched till acknowledge*)

IF ro_perOut < ri_chSP[1]AND NOT(wo_alarmOut.3 OR wo_alarmOut.4) THEN x_alarm2Temp1 := 1; ELSE x_alarm2Temp1 := 0; END_IF
ton_delay2(IN:= x_alarm2Temp1 AND NOT wi_chPara.1 AND NOT wi_chParaJm.1, PT:= REAL_TO_TIME ( ri_chSP[4]*1000), Q=> wo_alarmOut.1, ET=> );(*Level 2 alarm steady*)
tp_almPulse2(IN:=wo_alarmOut.1 , PT:= T#1s, Q=> w_alarmOutp_temp.1, ET=> );(*Level 2 alarm single pulse*)
IF (w_alarmOutp_temp.1 OR wo_alarmOutp.1) AND NOT xi_ack THEN wo_alarmOutp.1:=1; ELSE wo_alarmOutp.1:=0; END_IF(*Level 1 alarm single pulse latched till acknowledge*)

IF ro_perOut > ri_chSP[2] THEN x_alarm3Temp1 := 1; ELSE x_alarm3Temp1 := 0; END_IF
ton_delay3(IN:= x_alarm3Temp1 AND NOT wi_chPara.2 AND NOT wi_chParaJm.2, PT:= REAL_TO_TIME ( ri_chSP[5]*1000), Q=> wo_alarmOut.2, ET=> );(*Level 3 alarm steady*)
tp_almPulse3(IN:=wo_alarmOut.2 , PT:= T#1s, Q=> w_alarmOutp_temp.2, ET=> );(*Level 3 alarm single pulse*)
IF (w_alarmOutp_temp.2 OR wo_alarmOutp.2) AND NOT xi_ack THEN wo_alarmOutp.2:=1; ELSE wo_alarmOutp.2:=0; END_IF(*Level 1 alarm single pulse latched till acknowledge*)

IF r_sensorValtemp < 3 THEN x_alarm4Temp1 := 1; ELSE x_alarm4Temp1 := 0; END_IF
ton_delay4(IN:= x_alarm4Temp1 AND NOT wi_chPara.3 AND NOT wi_chParaJm.3, PT:= REAL_TO_TIME ( ri_chSP[6]*1000), Q=> wo_alarmOut.3, ET=> );(*cable break alarm steady*)
tp_almPulse4(IN:=wo_alarmOut.3 , PT:= T#1s, Q=> w_alarmOutp_temp.3, ET=> );(*cable break alarm single pulse*)
IF (w_alarmOutp_temp.3 OR wo_alarmOutp.3) AND NOT xi_ack THEN wo_alarmOutp.3:=1; ELSE wo_alarmOutp.3:=0; END_IF(*cable break alarm single pulse latched till acknowledge*)

IF r_sensorValtemp >= 22 THEN x_alarm5Temp1 := 1; ELSE x_alarm5Temp1 := 0; END_IF
ton_delay5(IN:= x_alarm5Temp1 AND NOT wi_chPara.4 AND NOT wi_chParaJm.4, PT:= REAL_TO_TIME ( ri_chSP[6]*1000), Q=> wo_alarmOut.4, ET=> );(*over range alarm steady*)
tp_almPulse5(IN:=wo_alarmOut.4 , PT:= T#1s, Q=> w_alarmOutp_temp.4, ET=> );(*over range alarm single pulse*)
IF (w_alarmOutp_temp.4 OR wo_alarmOutp.4) AND NOT xi_ack THEN wo_alarmOutp.4:=1; ELSE wo_alarmOutp.4:=0; END_IF(*over range alarm single pulse latched till acknowledge*)

IF ro_perOut > ri_chSP[13] THEN x_alarm6Temp1 := 1; ELSE x_alarm6Temp1 := 0; END_IF
ton_delay6(IN:= x_alarm6Temp1 AND NOT wi_chPara.10 AND NOT wi_chParaJm.10, PT:= REAL_TO_TIME ( ri_chSP[14]*1000), Q=> wo_alarmOut.5, ET=> );(*Level 4 alarm steady*)
tp_almPulse6(IN:=wo_alarmOut.5 , PT:= T#1s, Q=> w_alarmOutp_temp.5, ET=> );(*Level 4 alarm single pulse*)
IF (w_alarmOutp_temp.5 OR wo_alarmOutp.5) AND NOT xi_ack THEN wo_alarmOutp.5:=1; ELSE wo_alarmOutp.5:=0; END_IF(*Level 4 alarm single pulse latched till acknowledge*)

(*Alarm message*)
IF	wo_alarmOut.0 AND  wo_alarmOut.1 AND NOT wo_alarmOut.3 AND NOT wo_alarmOut.4 AND NOT xi_comErr  THEN	wo_alarmMsg :=1;(*LoLo*)
ELSE IF	NOT wo_alarmOut.0 AND wo_alarmOut.1 AND NOT wo_alarmOut.3 AND NOT wo_alarmOut.4 AND NOT xi_comErr THEN	wo_alarmMsg :=2;(*Lo*)
ELSE IF	NOT wo_alarmOut.5 AND wo_alarmOut.2 AND NOT wo_alarmOut.3 AND NOT wo_alarmOut.4 AND NOT xi_comErr THEN	wo_alarmMsg :=3;(*Hi*)
ELSE IF	wo_alarmOut.5 AND wo_alarmOut.2 AND NOT wo_alarmOut.3 AND NOT wo_alarmOut.4 AND NOT xi_comErr THEN	wo_alarmMsg :=4;(*HiHi*)
ELSE IF	wo_alarmOut.3 OR wo_alarmOut.4 OR xi_comErr THEN	wo_alarmMsg :=5;(*Sensor fault*)
ELSE wo_alarmMsg :=0;	END_IF	END_IF	END_IF	END_IF	END_IF
(*common buzzer out*)
xo_buzPulse := (w_alarmOutp_temp.0 AND NOT wi_chPara.5) OR (w_alarmOutp_temp.1 AND NOT wi_chPara.6) OR (w_alarmOutp_temp.2 AND NOT wi_chPara.7) OR (w_alarmOutp_temp.3 AND NOT wi_chPara.8) OR (w_alarmOutp_temp.4 AND NOT wi_chPara.9) OR (w_alarmOutp_temp.5 AND NOT wi_chPara.11);
(*common indication*)
xo_ind :=wo_alarmOut.0 OR wo_alarmOut.1 OR wo_alarmOut.2 OR wo_alarmOut.3 OR wo_alarmOut.4 OR wo_alarmOut.5;
(*Total inhibited alarms from Jmobile*)
wo_inhTot := BOOL_TO_WORD(wi_chParaJm.0) + BOOL_TO_WORD(wi_chParaJm.1) + BOOL_TO_WORD(wi_chParaJm.2)
 + BOOL_TO_WORD(wi_chParaJm.3) + BOOL_TO_WORD(wi_chParaJm.4) + BOOL_TO_WORD(wi_chParaJm.10);

END_FUNCTION_BLOCK

// Device/Application/fb_linScaleR
FUNCTION_BLOCK fb_linScaleR
VAR_INPUT
	input  	: REAL ;
	xmax  	: REAL ;
	xmin	: REAL ;
	ymax	:REAL ;
	ymin	:REAL ;
END_VAR
VAR_OUTPUT
	result 		: REAL;
	error : BOOL ;
END_VAR
VAR
	m : REAL ;
	denominator : REAL ;
	x : REAL;
	a: REAL;
END_VAR


IF xmin = xmax THEN
	result := ymin;
	error :=1;
ELSE
	result := (ymax - ymin) / (xmax - xmin) * (LIMIT(xmin, input, xmax) - xmin) + ymin;
	error :=0;
END_IF;

END_FUNCTION_BLOCK

// Device/Application/fb_nonLinScale20
FUNCTION_BLOCK fb_nonLinScale20
VAR_INPUT
	input  	: REAL ;
	xval 	:	ARRAY[0..20] OF WORD;
	yval	:	ARRAY[0..20] OF WORD;

END_VAR
VAR_OUTPUT
	result 		: REAL;
	error : BOOL ;
END_VAR
VAR
	xmax : WORD;
	xmin : WORD;
	ymax : WORD;
	ymin : WORD;

	LinScale1: fb_linScaleR;
END_VAR

IF input >= xval[0] AND input < xval[1] THEN
xmax :=xval[1];		xmin := xval[0];		ymax :=yval[1];		ymin := yval[0];

ELSE IF input >= xval[1] AND input < xval[2] THEN
xmax :=xval[2];		xmin := xval[1];		ymax :=yval[2];		ymin := yval[1];

ELSE IF input >= xval[2] AND input < xval[3] THEN
xmax :=xval[3];		xmin := xval[2];		ymax :=yval[3];		ymin := yval[2];

ELSE IF input >= xval[3] AND input < xval[4] THEN
xmax :=xval[4];		xmin := xval[3];		ymax :=yval[4];		ymin := yval[3];

ELSE IF input >= xval[4] AND input < xval[5] THEN
xmax :=xval[5];		xmin := xval[4];		ymax :=yval[5];		ymin := yval[4];

ELSE IF input >= xval[5] AND input < xval[6] THEN
xmax :=xval[6];		xmin := xval[5];		ymax :=yval[6];		ymin := yval[5];

ELSE IF input >= xval[6] AND input < xval[7] THEN
xmax :=xval[7];		xmin := xval[6];		ymax :=yval[7];		ymin := yval[6];

ELSE IF input >= xval[7] AND input < xval[8] THEN
xmax :=xval[8];		xmin := xval[7];		ymax :=yval[8];		ymin := yval[7];

ELSE IF input >= xval[8] AND input < xval[9] THEN
xmax :=xval[9];		xmin := xval[8];		ymax :=yval[9];		ymin := yval[8];

ELSE IF input >= xval[9] AND input < xval[10] THEN
xmax :=xval[10];		xmin := xval[9];		ymax :=yval[10];		ymin := yval[9];

ELSE IF input >= xval[10] AND input < xval[11] THEN
xmax :=xval[11];		xmin := xval[10];		ymax :=yval[11];		ymin := yval[10];


ELSE IF input >= xval[11] AND input < xval[12] THEN
xmax :=xval[12];		xmin := xval[11];		ymax :=yval[12];		ymin := yval[11];


ELSE IF input >= xval[12] AND input < xval[13] THEN
xmax :=xval[13];		xmin := xval[12];		ymax :=yval[13];		ymin := yval[12];


ELSE IF input >= xval[13] AND input < xval[14] THEN
xmax :=xval[14];		xmin := xval[13];		ymax :=yval[14];		ymin := yval[13];


ELSE IF input >= xval[14] AND input < xval[15] THEN
xmax :=xval[15];		xmin := xval[14];		ymax :=yval[15];		ymin := yval[14];


ELSE IF input >= xval[15] AND input < xval[16] THEN
xmax :=xval[16];		xmin := xval[15];		ymax :=yval[16];		ymin := yval[15];


ELSE IF input >= xval[16] AND input < xval[17] THEN
xmax :=xval[17];		xmin := xval[16];		ymax :=yval[17];		ymin := yval[16];


ELSE IF input >= xval[17] AND input < xval[18] THEN
xmax :=xval[18];		xmin := xval[17];		ymax :=yval[18];		ymin := yval[17];


ELSE IF input >= xval[18] AND input < xval[19] THEN
xmax :=xval[19];		xmin := xval[18];		ymax :=yval[19];		ymin := yval[18];


ELSE IF input >= xval[19] AND input <= xval[20] THEN
xmax :=xval[20];		xmin := xval[19];		ymax :=yval[20];		ymin := yval[19];

END_IF	END_IF	END_IF	END_IF	END_IF	END_IF	END_IF	END_IF	END_IF	END_IF
END_IF	END_IF	END_IF	END_IF	END_IF	END_IF	END_IF	END_IF	END_IF	END_IF

LinScale1(
	input:=input ,
	xmax:=REAL_TO_WORD(xmax) ,
	xmin:= REAL_TO_WORD(xmin),
	ymax:=REAL_TO_WORD(ymax) ,
	ymin:= REAL_TO_WORD(ymin),
	result=>result  ,
	error=> error);

END_FUNCTION_BLOCK

// Device/Application/sh_2
FUNCTION_BLOCK sh_2
VAR_INPUT
	in : REAL;
	PT : TIME;
	N : INT := 16;
	disc : INT;
END_VAR
VAR_OUTPUT
	out : REAL;
	trig : BOOL;
	avg : REAL;
	high: REAL;
	low: REAL;
END_VAR
VAR
	M : INT;
	buf : ARRAY[0..15] OF REAL;
	buf2 : ARRAY[0..15] OF REAL;
	last : TIME;
	i : INT;
	start: INT;
	temp: REAL;
	stop: INT;
	tx: TIME;
	d2: INT;
	even :BOOL;
END_VAR

(* read system time *)
tx := TIME();
d2 := SHR(disc,1);
even:= NOT disc.0;
IF tx - last >= PT THEN
	last := tx;
	trig := TRUE;

	(* limit M to 0..16 *)
	M := LIMIT(1,N,16);

	(* edge detected lets take the sample *)
	FOR i := M - 1 TO 1 BY -1 DO buf2[i] := buf2[i-1]; END_FOR;
	buf2[0] := in;
	out := in;
	buf := buf2;

	(* sort the ARRAY lowest value AT 0 *)
	FOR start := 0 TO M - 2 DO
		FOR i := start+1 TO M - 1 DO
			IF buf[start] > buf[i] THEN
				temp := buf[start];
				buf[start] := buf[i];
				buf[i] := temp;
			END_IF;
		END_FOR;
	END_FOR;

	(* any calculation with the samples is here *)
	stop := M - 1 - d2;
	start := d2;
	IF NOT even THEN start := start + 1; END_IF;
	avg := 0;
	FOR i := start TO stop DO avg := avg + buf[i]; END_FOR;
	avg := avg / INT_TO_REAL(stop - start +1);
	low := buf[start];
	high := buf[stop];
ELSE
	Trig := FALSE;
END_IF;

(* revision history
hm 20. jan. 2007	rev 1.1
	added input N to specify the amout of samples for average and high low calculations
	added trig output

hm 10. sep. 2007 	rev 1.2
	an error would be generated if N was set to 0, now n is forced to1 if set to 0.
	index was out of array.

hm	17. sep. 2007	rev 1.3
	replaced time() with t_plc_ms() for compatibility reasons

hm	6. jan. 2008	rev 1.4
	improved performance

hm	14. jun. 2008	rev 1.5
	set default for input N = 16

hm	10. mar. 2009	rev 1.6
	added type conversion for compatibility reasons

*)

END_FUNCTION_BLOCK

// Device/Application/fb_fluctDet
FUNCTION_BLOCK fb_fluctDet
VAR_INPUT
	ri_in : REAL;
	ri_rocVal: REAL;
	ri_sampTime: REAL :=0.5;
	ri_sholdT : REAL :=3.0;
END_VAR
VAR_OUTPUT
	xo_valFluct: BOOL;
END_VAR
VAR
	M : INT;
	buf : ARRAY[0..4] OF REAL;
	j : WORD;
	TONblink: TON;
	TPblink: TP;
	N: INT;
	CTU1: CTU;
	TONrst: TON;
	dif1: REAL;
	dif2: REAL;
	dif3: REAL;
	dif4: REAL;

	valFluct: BOOL;

	tcFilt: TIME;
END_VAR


TONblink(IN:=NOT TPblink.Q , PT:=REAL_TO_TIME ( ri_sampTime*1000) , Q=> , ET=> );
TPblink(IN:=TONblink.Q , PT:= T#500ms, Q=> , ET=> );
CTU1(
	CU:=TPblink.Q ,
	RESET:= CTU1.Q,
	PV:= 4,
	Q=> , 
	CV=> );
j:=CTU1.CV;
buf[j] := ri_in;

IF (buf[1]- buf[0]) > 0 THEN dif1 := buf[1]- buf[0]; ELSE dif1 := -(buf[1]- buf[0]); END_IF
IF (buf[2]- buf[1]) > 0 THEN dif2 := buf[2]- buf[1]; ELSE dif2 := -(buf[2]- buf[1]); END_IF
IF (buf[3]- buf[2]) > 0 THEN dif3 := buf[3]- buf[2]; ELSE dif3 := -(buf[3]- buf[2]); END_IF
IF (buf[4]- buf[3]) > 0 THEN dif4 := buf[4]- buf[3]; ELSE dif4 := -(buf[4]- buf[3]); END_IF

TONrst(IN:= NOT valFluct , PT:=REAL_TO_TIME ( ri_sholdT*1000) , Q=> , ET=> );

IF (dif1 > ri_rocVal) OR (dif2 > ri_rocVal) OR(dif3 > ri_rocVal) OR(dif4 > ri_rocVal) THEN valFluct :=1; ELSE valFluct :=0; END_IF

IF (valFluct OR xo_valFluct) AND NOT TONrst.Q THEN xo_valFluct :=1; ELSE  xo_valFluct :=0;  END_IF

END_FUNCTION_BLOCK

// Device/Application/fb_buzzer
FUNCTION_BLOCK fb_buzzer
VAR_INPUT
	Lwi_AlarmBuzzer: WORD;
	Lwi_AlarmInd: WORD;
	LDi_Ack: BOOL;
END_VAR
VAR_OUTPUT
	LDo_Acoustic: BOOL;
	LDo_Visual: BOOL;
END_VAR
VAR
	AlarmBuzzer: BOOL;
	AlarmInd: BOOL;
	TONblink: TON;
	TPblink: TP;
END_VAR

IF Lwi_AlarmBuzzer.0 OR Lwi_AlarmBuzzer.1 OR Lwi_AlarmBuzzer.2 OR Lwi_AlarmBuzzer.3 OR Lwi_AlarmBuzzer.4 OR Lwi_AlarmBuzzer.5 OR Lwi_AlarmBuzzer.6 OR Lwi_AlarmBuzzer.7
OR Lwi_AlarmBuzzer.8 OR Lwi_AlarmBuzzer.9 OR Lwi_AlarmBuzzer.10 OR Lwi_AlarmBuzzer.11 OR Lwi_AlarmBuzzer.12 OR Lwi_AlarmBuzzer.13
OR Lwi_AlarmBuzzer.14 OR Lwi_AlarmBuzzer.15 THEN
AlarmBuzzer:= 1;
ELSE
AlarmBuzzer:= 0;
END_IF

IF Lwi_AlarmInd.0 OR Lwi_AlarmInd.1 OR Lwi_AlarmInd.2 OR Lwi_AlarmInd.3 OR Lwi_AlarmInd.4 OR Lwi_AlarmInd.5 OR Lwi_AlarmInd.6 OR Lwi_AlarmInd.7
OR Lwi_AlarmInd.8 OR Lwi_AlarmInd.9 OR Lwi_AlarmInd.10 OR Lwi_AlarmInd.11 OR Lwi_AlarmInd.12 OR Lwi_AlarmInd.13
OR Lwi_AlarmInd.14 OR Lwi_AlarmInd.15 THEN
AlarmInd:= 1;
ELSE
AlarmInd:= 0;
END_IF

IF (AlarmBuzzer OR LDo_Acoustic) AND NOT LDi_Ack THEN
LDo_Acoustic	:=	1;
ELSE
LDo_Acoustic	:=	0;
END_IF

TONblink(IN:=NOT TPblink.Q AND LDo_Acoustic , PT:=T#1s , Q=> , ET=> );

TPblink(IN:=TONblink.Q AND LDo_Acoustic , PT:= T#1s, Q=> , ET=> );

LDo_Visual	:=	AlarmInd AND NOT TPblink.Q;

END_FUNCTION_BLOCK

// Device/Application/fb_comAlarm
FUNCTION_BLOCK fb_comAlarm
VAR_INPUT
	LDi_Accoustic1: BOOL;
	LDi_Accoustic2: BOOL;
	LDi_Accoustic3: BOOL;
	LDi_Visual1: BOOL;
	LDi_Visual2: BOOL;
	LDi_Visual3: BOOL;

	LDi_BuzStop1:BOOL;
	LDi_BuzStop2:BOOL;
	LDi_BuzStop3:BOOL;
	LDi_BuzStop4: BOOL;
	LDi_Ack1: BOOL;
	LDi_Ack2: BOOL;
	LDi_Ack3: BOOL;
	LDi_Ack4: BOOL;
END_VAR
VAR_OUTPUT
	LDo_Accoustic1: BOOL;
	LDo_Accoustic2: BOOL;
	LDo_Visual1: BOOL;
	LDo_Visual2: BOOL;
	LDo_BuzStop: BOOL;
	LDo_Ack: BOOL;
END_VAR
VAR
END_VAR

IF LDi_Accoustic1 OR LDi_Accoustic2 OR LDi_Accoustic3 THEN
LDo_Accoustic1 := 1;
LDo_Accoustic2 := 1;
ELSE
LDo_Accoustic1 := 0;
LDo_Accoustic2 := 0;
END_IF

IF LDi_Visual1 OR LDi_Visual2 OR LDi_Visual3 THEN
LDo_Visual1 := 1;
LDo_Visual2 := 1;
ELSE
LDo_Visual1 := 0;
LDo_Visual2 := 0;
END_IF

IF 	LDi_BuzStop1 OR LDi_BuzStop2 OR LDi_BuzStop3 OR LDi_BuzStop4 THEN
LDo_BuzStop := 1;
ELSE
LDo_BuzStop := 0;
END_IF

IF LDi_Ack1 OR LDi_Ack2 OR LDi_Ack3 OR LDi_Ack4 THEN
LDo_Ack := 1;
ELSE
LDo_Ack := 0;
END_IF

END_FUNCTION_BLOCK

// Device/Application/commCheck
FUNCTION_BLOCK commCheck
VAR_INPUT
	Lbi_Enable: BOOL;
	Lbi_Resp1: BOOL;
	Lbi_Resp2: BOOL;
	Lbi_Resp3: BOOL;
	Lbi_Resp4: BOOL;
END_VAR
VAR_OUTPUT
	Lbo_Request: BOOL;
	Lbo_ComErr1: BOOL;
	Lbo_ComErr2: BOOL;
	Lbo_ComErr3: BOOL;
	Lbo_ComErr4: BOOL;
END_VAR
VAR
	Lto_ComErr1: BOOL;
	Lto_ComErr2: BOOL;
	Lto_ComErr3: BOOL;
	Lto_ComErr4: BOOL;
	TOF1: TOF;
	TP1: TP;
	TON1a: TON;
	TON1b: TON;
	TON2a: TON;
	TON2b: TON;
	TON3a: TON;
	TON3b: TON;
	TON4a: TON;
	TON4b: TON;

END_VAR

TOF1(IN:=TP1.Q  AND Lbi_Enable , PT:=T#1S , Q=> , ET=> );

TP1(IN:=NOT TOF1.Q  AND Lbi_Enable , PT:=T#1s , Q=> , ET=> );

Lbo_Request := TP1.Q;

TON1a(IN:= NOT Lbi_Resp1 , PT:=T#4s , Q=> , ET=> );
TON1b(IN:=Lbi_Resp1 , PT:=T#4s , Q=> , ET=> );
Lto_ComErr1:= TON1a.Q OR TON1b.Q;
Lbo_ComErr1:= NOT Lto_ComErr1;

TON2a(IN:= NOT Lbi_Resp2 , PT:=T#4s , Q=> , ET=> );
TON2b(IN:=Lbi_Resp2 , PT:=T#4s , Q=> , ET=> );
Lto_ComErr2:= TON2a.Q OR TON2b.Q;
Lbo_ComErr2:= NOT Lto_ComErr2;

TON3a(IN:= NOT Lbi_Resp3 , PT:=T#4s , Q=> , ET=> );
TON3b(IN:=Lbi_Resp3 , PT:=T#4s , Q=> , ET=> );
Lto_ComErr3:= TON3a.Q OR  TON3b.Q;
Lbo_ComErr3:= NOT Lto_ComErr3;

TON4a(IN:= NOT Lbi_Resp4 , PT:=T#2s , Q=> , ET=> );
TON4b(IN:=Lbi_Resp4 , PT:=T#2s , Q=> , ET=> );
Lto_ComErr4:= TON4a.Q OR  TON4b.Q;
Lbo_ComErr4:= NOT Lto_ComErr4;

END_FUNCTION_BLOCK

// Device/Application/fb_scaling20R
FUNCTION_BLOCK fb_scaling20R
VAR_INPUT
	
	ii_pts	:	INT;
	ri_input	:	REAL;
	ri_xval 	:	ARRAY[1..20] OF REAL;
	ri_yval	:	ARRAY[1..20] OF REAL;
END_VAR
VAR_OUTPUT
	ro_result: REAL;
END_VAR
VAR
	j	:	INT;
	xmax : REAL;
	xmin : REAL;
	ymax : REAL;
	ymin : REAL;
	error: BOOL;
END_VAR

j:=2;

WHILE j< ii_pts AND (ri_xval[j] < ri_input) DO
j:=j+1;
END_WHILE

xmax :=ri_xval[j];		
xmin := ri_xval[j-1];		
ymax :=ri_yval[j];		
ymin := ri_yval[j-1];

IF xmin = xmax THEN
	ro_result := ymin;
	error :=1;
ELSE
	(*ro_result := (ymax - ymin) / (xmax - xmin) * (input - xmin) + ymin;*)(*input not limited*)
	ro_result := (((ymax - ymin) / (xmax - xmin)) * (LIMIT(xmin, ri_input, xmax) - xmin)) + ymin;(*input limited to scaling min and max range*)
	error :=0;
END_IF;

END_FUNCTION_BLOCK

// Device/Application/fb_h2s
FUNCTION_BLOCK fb_h2s
VAR_INPUT
	wi_sensorVal	: WORD;
	wi_chPara	: WORD;(*0:inhL1, 1:inhL2, 2:inhL3, 3:inhCable break, 4:inhOver range, 5:buz en L1, 6:buz en L2, 7:buz en L3, 8:buz en err1, 9:buz en err2, 10:inhL4, 11:buz en L4, 12: Auto filter enable
							13:Fill input sensor min value and range when tank empty, 14: Fill input sensor max value and range when tank full*)
	wi_chParaJm	: WORD;
	xi_comErr	:BOOL;
	xi_ack	:BOOL;
END_VAR
VAR_OUTPUT
	ro_perOut	:REAL;
	ro_curOut	:REAL;
	wo_alarmOut	 : WORD;(*alarm out steady*)
	wo_alarmOutp	 : WORD;(*alarm out single pulse latched till acknowledge*)
	xo_buzPulse	: BOOL;
	xo_ind	:BOOL;
	xo_buzPulse1	: BOOL;
	xo_ind1	:BOOL;
	wo_alarmMsg	:WORD;(*Alarm msg*)
	wo_inhTot :WORD;	
END_VAR
VAR
	r_sensorValtemp0 : REAL;
	r_sensorValtemp1 : REAL;
	r_sensorValtemp2 : REAL;
	r_sensorValtemp3 : REAL;
	r_sensorVal	: REAL;
	r_sensorValtemp	:REAL;
	w_alarmOutp_temp	 : WORD;
	ton_delay1	:TON;
	ton_delay2	:TON;
	ton_delay3	:TON;
	ton_delay4	:TON;
	ton_delay5	:TON;

	tp_almPulse1	:TP;
	tp_almPulse2	:TP;
	tp_almPulse3	:TP;
	tp_almPulse4	:TP;
	tp_almPulse5	:TP;

	x_alarm1Temp1	:BOOL;
	x_alarm2Temp1	:BOOL;
	x_alarm3Temp1	:BOOL;
	x_alarm4Temp1	:BOOL;
	x_alarm5Temp1	:BOOL;
	x_alarm6Temp1	:BOOL;
	LinScale1: fb_linScaleR;

	r_valOut: REAL;
	filter_SH2: sh_2;

END_VAR
VAR_IN_OUT
	ri_chSP	: ARRAY[0..23] OF REAL;(*0:L1Lt, 1:L2Lt, 2:L3Lt, 3:L1delay, 4:L2delay, 5:L3delay,6:Errdelay,
											7:ErrFactor, 8:SensorValMin,9:SensorValMax, 10:SensorRangeMin, 11:SensorRangeMax, 12:filterVal, 
											13:L4Lt, 14:L4delay, 15:heightMin, 16:heightMax, 17:density, 18:unusable , 19:height offset in mm, 
											Auto filter-->20: rate of change, 21: sampling time, 22:sample hold time, 23:filter time constant*)
END_VAR


filter_SH2(
	in:=wi_sensorVal ,
	PT:= REAL_TO_TIME ( ri_chSP[12]*1000),
	N:= 16,
	disc:=0 ,
	out=> r_sensorValtemp1,
	trig=> ,
	avg=> r_sensorValtemp0,
	high=> ,
	low=> );
IF (ri_chSP[12] > 0) THEN r_sensorValtemp2:= r_sensorValtemp0; ELSE r_sensorValtemp2:= r_sensorValtemp1; END_IF

IF  r_sensorValtemp1 = 3 THEN r_sensorValtemp3 := 0; ELSE r_sensorValtemp3 :=  r_sensorValtemp2; END_IF(*return to 0 incase of cable break*)
ro_curOut :=  (20 * r_sensorValtemp3)/4095;(*-->convert  A/D row value to mA-->for 0-20mA input-->	ro_curOut := (20 - 0) / (32760 - 0) * (r_sensorValtemp3 - 0) + 0;*)
(*-->convert  A/D row value to mA-->for 4-20mA input-->	ro_curOut := (20 - 4) / (32760 - 0) * (r_sensorValtemp3 - 0) + 4;*)
r_sensorValtemp := ro_curOut* ri_chSP[7]; (*eror compensation*)
(*method 2 calibration*)

(*scale to output value as per output range given*)
LinScale1(
	input:= r_sensorValtemp,
	xmax:= ri_chSP[9],
	xmin:= ri_chSP[8],
	ymax:= ri_chSP[11],
	ymin:= ri_chSP[10],
	result=> ro_perOut,
	error=> );

(*Alarms : level1, level2, ;evel3, cable break, over range, level4*)
IF ro_perOut >= ri_chSP[0] AND NOT (wo_alarmOut.3 OR wo_alarmOut.4) THEN x_alarm1Temp1 := 1; ELSE x_alarm1Temp1 := 0; END_IF
ton_delay1(IN:= x_alarm1Temp1 AND NOT wi_chPara.0 AND NOT wi_chParaJm.0, PT:= REAL_TO_TIME ( ri_chSP[3]*1000), Q=> wo_alarmOut.0, ET=> );(*Level 1 alarm steady*)
tp_almPulse1(IN:=wo_alarmOut.0 , PT:= T#1s, Q=> w_alarmOutp_temp.0, ET=> );(*Level 1 alarm single pulse*)
IF (w_alarmOutp_temp.0 OR wo_alarmOutp.0) AND NOT xi_ack THEN wo_alarmOutp.0:=1; ELSE wo_alarmOutp.0:=0; END_IF(*Level 1 alarm single pulse latched till acknowledge*)

IF ro_perOut >= ri_chSP[1] AND NOT (wo_alarmOut.3 OR wo_alarmOut.4)THEN x_alarm2Temp1 := 1; ELSE x_alarm2Temp1 := 0; END_IF
ton_delay2(IN:= x_alarm2Temp1 AND NOT wi_chPara.1 AND NOT wi_chParaJm.1, PT:= REAL_TO_TIME ( ri_chSP[4]*1000), Q=> wo_alarmOut.1, ET=> );(*Level 2 alarm steady*)
tp_almPulse2(IN:=wo_alarmOut.1 , PT:= T#1s, Q=> w_alarmOutp_temp.1, ET=> );(*Level 2 alarm single pulse*)
IF (w_alarmOutp_temp.1 OR wo_alarmOutp.1) AND NOT xi_ack THEN wo_alarmOutp.1:=1; ELSE wo_alarmOutp.1:=0; END_IF(*Level 1 alarm single pulse latched till acknowledge*)

IF ro_perOut >= ri_chSP[2]AND NOT (wo_alarmOut.3 OR wo_alarmOut.4) THEN x_alarm3Temp1 := 1; ELSE x_alarm3Temp1 := 0; END_IF
ton_delay3(IN:= x_alarm3Temp1 AND NOT wi_chPara.2 AND NOT wi_chParaJm.2, PT:= REAL_TO_TIME ( ri_chSP[5]*1000), Q=> wo_alarmOut.2, ET=> );(*Level 3 alarm steady*)
tp_almPulse3(IN:=wo_alarmOut.2 , PT:= T#1s, Q=> w_alarmOutp_temp.2, ET=> );(*Level 3 alarm single pulse*)
IF (w_alarmOutp_temp.2 OR wo_alarmOutp.2) AND NOT xi_ack THEN wo_alarmOutp.2:=1; ELSE wo_alarmOutp.2:=0; END_IF(*Level 1 alarm single pulse latched till acknowledge*)

IF r_sensorValtemp < 3 THEN x_alarm4Temp1 := 1; ELSE x_alarm4Temp1 := 0; END_IF
ton_delay4(IN:= x_alarm4Temp1 AND NOT wi_chPara.3 AND NOT wi_chParaJm.3, PT:= REAL_TO_TIME ( ri_chSP[6]*1000), Q=> wo_alarmOut.3, ET=> );(*cable break alarm steady*)
tp_almPulse4(IN:=wo_alarmOut.3 , PT:= T#1s, Q=> w_alarmOutp_temp.3, ET=> );(*cable break alarm single pulse*)
IF (w_alarmOutp_temp.3 OR wo_alarmOutp.3) AND NOT xi_ack THEN wo_alarmOutp.3:=1; ELSE wo_alarmOutp.3:=0; END_IF(*cable break alarm single pulse latched till acknowledge*)

IF r_sensorValtemp >= 22 THEN x_alarm5Temp1 := 1; ELSE x_alarm5Temp1 := 0; END_IF
ton_delay5(IN:= x_alarm5Temp1 AND NOT wi_chPara.4 AND NOT wi_chParaJm.4, PT:= REAL_TO_TIME ( ri_chSP[6]*1000), Q=> wo_alarmOut.4, ET=> );(*over range alarm steady*)
tp_almPulse5(IN:=wo_alarmOut.4 , PT:= T#1s, Q=> w_alarmOutp_temp.4, ET=> );(*over range alarm single pulse*)
IF (w_alarmOutp_temp.4 OR wo_alarmOutp.4) AND NOT xi_ack THEN wo_alarmOutp.4:=1; ELSE wo_alarmOutp.4:=0; END_IF(*over range alarm single pulse latched till acknowledge*)



(*Alarm message*)
IF	wo_alarmOut.0 AND NOT wo_alarmOut.1 AND NOT wo_alarmOut.2 AND NOT wo_alarmOut.3 AND NOT wo_alarmOut.4 AND NOT xi_comErr  THEN	wo_alarmMsg :=1;(*LoLo*)
ELSE IF	wo_alarmOut.0 AND wo_alarmOut.1 AND NOT wo_alarmOut.2 AND NOT wo_alarmOut.3 AND NOT wo_alarmOut.4 AND NOT xi_comErr THEN	wo_alarmMsg :=2;(*Lo*)
ELSE IF	wo_alarmOut.0 AND wo_alarmOut.1 AND wo_alarmOut.2 AND NOT wo_alarmOut.3 AND NOT wo_alarmOut.4 AND NOT xi_comErr THEN	wo_alarmMsg :=3;(*Hi*)
(*ELSE IF	wo_alarmOut.5 AND wo_alarmOut.2 AND NOT wo_alarmOut.3 AND NOT wo_alarmOut.4 AND NOT xi_comErr THEN	wo_alarmMsg :=4;(*HiHi*)*)
ELSE IF	wo_alarmOut.3 OR wo_alarmOut.4 OR xi_comErr THEN	wo_alarmMsg :=5;(*Sensor fault*)
ELSE wo_alarmMsg :=0;	END_IF	END_IF	END_IF	END_IF	(*END_IF*)
(*common buzzer out*)
xo_buzPulse := (w_alarmOutp_temp.0 AND NOT wi_chPara.5) OR (w_alarmOutp_temp.1 AND NOT wi_chPara.6) OR (w_alarmOutp_temp.2 AND NOT wi_chPara.7) OR (w_alarmOutp_temp.3 AND NOT wi_chPara.8) OR (w_alarmOutp_temp.4 AND NOT wi_chPara.9) OR (w_alarmOutp_temp.5 AND NOT wi_chPara.11);
(*common indication*)
xo_ind :=wo_alarmOut.0 OR wo_alarmOut.1 OR wo_alarmOut.2 OR wo_alarmOut.3 OR wo_alarmOut.4 OR wo_alarmOut.5;
(*Level 2 alarm out to H2s buzzer*)
xo_buzPulse1:= (w_alarmOutp_temp.1 AND NOT wi_chPara.6);
xo_ind1:= wo_alarmOut.1;
(*Total inhibited alarms from Jmobile*)
wo_inhTot := BOOL_TO_WORD(wi_chParaJm.0) + BOOL_TO_WORD(wi_chParaJm.1) + BOOL_TO_WORD(wi_chParaJm.2)
 + BOOL_TO_WORD(wi_chParaJm.3) + BOOL_TO_WORD(wi_chParaJm.4);

END_FUNCTION_BLOCK

// Device/Application/fb_tankMonitor_magLt
FUNCTION_BLOCK fb_tankMonitor_magLt
VAR_INPUT
	wi_sensorVal	: WORD;
	wi_samplingIn	: ARRAY[0..20] OF  WORD;
	wi_samplingOut	: ARRAY[0..20] OF  WORD;

	wi_chPara	: WORD;(*0:inhL1, 1:inhL2, 2:inhL3, 3:inhCable break, 4:inhOver range, 5:buz en L1, 6:buz en L2, 7:buz en L3, 8:buz en err1, 9:buz en err2, 10:inhL4, 11:buz en L4, 12: Auto filter enable
							13:Fill input sensor min value and range when tank empty, 14: Fill input sensor max value and range when tank full*)
	wi_chParaJm	: WORD;	
	xi_comErr	:BOOL;
	xi_ack	:BOOL;
END_VAR
VAR_OUTPUT
	ro_pressOut	:REAL;
	ro_htOut	:REAL;
	ro_volOut	:REAL;
	ro_perOut	:REAL;
	ro_curOut	:REAL;
	wo_alarmOut	 : WORD;(*alarm out steady*)
	wo_alarmOutp	 : WORD;(*alarm out single pulse latched till acknowledge*)
	xo_buzPulse	: BOOL;
	xo_ind	:BOOL;
	wo_alarmMsg	:WORD;(*Alarm msg*)
	wo_inhTot :WORD;
END_VAR
VAR
	r_sensorValtemp0 : REAL;
	r_sensorValtemp1 : REAL;
	r_sensorValtemp2 : REAL;
	r_sensorValtemp3 : REAL;
	r_sensorVal	: REAL;
	r_sensorValtemp	:REAL;
	w_alarmOutp_temp	 : WORD;
	ton_delay1	:TON;
	ton_delay2	:TON;
	ton_delay3	:TON;
	ton_delay4	:TON;
	ton_delay5	:TON;
	ton_delay6	:TON;
	tp_almPulse1	:TP;
	tp_almPulse2	:TP;
	tp_almPulse3	:TP;
	tp_almPulse4	:TP;
	tp_almPulse5	:TP;
	tp_almPulse6	:TP;
	x_alarm1Temp1	:BOOL;
	x_alarm2Temp1	:BOOL;
	x_alarm3Temp1	:BOOL;
	x_alarm4Temp1	:BOOL;
	x_alarm5Temp1	:BOOL;
	x_alarm6Temp1	:BOOL;
	LinScale1: fb_linScaleR;
	LinScale2: fb_linScaleR;
	r_valOut: REAL;
	r_pressOut: REAL;
	NonLinScale1: fb_nonLinScale20;
	r_volOut	:REAL;
	r_volOut1	:REAL;
	r_htOut	:REAL;
	r_htOut1	:REAL;
	linScale_r0: fb_linScaleR;
	filter_SH2: sh_2;
	fluctDet1: fb_fluctDet;
END_VAR
VAR_IN_OUT
	ri_chSP	: ARRAY[0..23] OF REAL;(*0:L1Lt, 1:L2Lt, 2:L3Lt, 3:L1delay, 4:L2delay, 5:L3delay,6:Errdelay,
											7:ErrFactor, 8:SensorValMin,9:SensorValMax, 10:SensorRangeMin, 11:SensorRangeMax, 12:filterVal, 
											13:L4Lt, 14:L4delay, 15:heightMin, 16:heightMax, 17:density, 18:unusable , 19:height offset in mm, 
											Auto filter-->20: rate of change, 21: sampling time, 22:sample hold time, 23:filter time constant*)
END_VAR

(*fb_tankMonitor_magLt: for magnetic float level transmitter-06Jan2021*)
(*fluctDet1(ri_in:=wi_sensorVal , wi_setVal:=1020 , xo_valFluct=> );*)
fluctDet1(
	ri_in:=wi_sensorVal ,
	ri_rocVal:= ri_chSP[20],
	ri_sampTime:= ri_chSP[21],
	ri_sholdT:=ri_chSP[22] ,
	xo_valFluct=> );
IF fluctDet1.xo_valFluct AND wi_chPara.12 THEN filter_SH2.PT := REAL_TO_TIME ( ri_chSP[23]*1000); ELSE filter_SH2.PT :=REAL_TO_TIME ( ri_chSP[12]*1000); END_IF
filter_SH2(
	in:=wi_sensorVal ,
	PT:= ,
	N:= 16,
	disc:=0 ,
	out=> r_sensorValtemp1,
	trig=> ,
	avg=> r_sensorValtemp0,
	high=> ,
	low=> );
IF (fluctDet1.xo_valFluct AND wi_chPara.12) OR (ri_chSP[12] > 0) THEN r_sensorValtemp2:= r_sensorValtemp0; ELSE r_sensorValtemp2:= r_sensorValtemp1; END_IF

IF  r_sensorValtemp1 = 3 THEN r_sensorValtemp3 := 0; ELSE r_sensorValtemp3 :=  r_sensorValtemp2; END_IF(*return to 0 incase of cable break*)
ro_curOut :=  (20 * r_sensorValtemp3)/4095;(*-->convert  A/D row value to mA-->for 0-20mA input-->	ro_curOut := (20 - 0) / (32760 - 0) * (r_sensorValtemp3 - 0) + 0;*)
(*-->convert  A/D row value to mA-->for 4-20mA input-->	ro_curOut := (20 - 4) / (32760 - 0) * (r_sensorValtemp3 - 0) + 4;*)
r_sensorValtemp := ro_curOut* ri_chSP[7]; (*eror compensation*)
(*method 2 calibration*)

IF wi_chPara.13 THEN ri_chSP[8]:=r_sensorValtemp; ri_chSP[10]:=(ri_chSP[15] * ri_chSP[17] * 9.8066)/1000; END_IF(*Tank empty set*)
IF wi_chPara.14 THEN ri_chSP[9]:=r_sensorValtemp; ri_chSP[11]:=(ri_chSP[16] * ri_chSP[17] * 9.8066)/1000; END_IF(*Tank full set*)
(*scale to output value as per output range given*)
LinScale1(
	input:= r_sensorValtemp,
	xmax:= ri_chSP[9],
	xmin:= ri_chSP[8],
	ymax:= ri_chSP[11],
	ymin:= ri_chSP[10],
	result=> r_htOut1(*r_pressOut*), (*For magnetic float LT input mA to be scaled to height*)
	error=> );
ro_pressOut:=0 ; (*For magnetic float LT input mA to be scaled to height. No pressure involved*)
(*
(*Liquid height = Pressure / ( Liquid density * Gravity)          -> Pressure in pascal*)
IF ri_chSP[17] > 0 THEN
r_htOut1 := (ro_pressOut * 1000) / (ri_chSP[17] *9.8066);(*height in mm*)
ELSE r_htOut1 :=0; END_IF*)

IF r_htOut1 > 10 AND ri_chSP[19] > 0 THEN r_htOut := r_htOut1 + ri_chSP[19];(*Added height +offset in mm*)
ELSE IF r_htOut1 >= -ri_chSP[19] AND ri_chSP[19] < 0 THEN r_htOut := r_htOut1 + ri_chSP[19];(*Added height -offset in mm*)
ELSE IF r_htOut1 < -ri_chSP[19] AND ri_chSP[19] < 0 THEN r_htOut := 0;(*Added height -offset in mm*)
ELSE r_htOut := r_htOut1; END_IF END_IF END_IF
IF r_htOut > ri_chSP[16] THEN ro_htOut:=ri_chSP[16];(*Limited to max height*)
ELSE ro_htOut:=r_htOut ; END_IF
(*scale to percentage of height *)
LinScale2(
	input:= ro_htOut,
	xmax:= ri_chSP[16],
	xmin:= ri_chSP[15],
	ymax:= 100,
	ymin:= 0,
	result=> ro_perOut,
	error=> );
(*scale as per sounding table*)
NonLinScale1(
	input:=ro_htOut ,
	xval:=wi_samplingIn ,
	yval:= wi_samplingOut,
	result=>r_volOut ,
	error=> );
IF r_volOut <= ri_chSP[18] AND  ri_chSP[18] > 0  THEN r_volOut1 := 0;
ELSE r_volOut1 :=  r_volOut - ri_chSP[18]; END_IF
ro_volOut	:= r_volOut1;
(*Alarms : level1, level2, ;evel3, cable break, over range, level4*)
IF ro_perOut < ri_chSP[0]AND NOT(wo_alarmOut.3 OR wo_alarmOut.4) THEN x_alarm1Temp1 := 1; ELSE x_alarm1Temp1 := 0; END_IF
ton_delay1(IN:= x_alarm1Temp1 AND NOT wi_chPara.0 AND NOT wi_chParaJm.0, PT:= REAL_TO_TIME ( ri_chSP[3]*1000), Q=> wo_alarmOut.0, ET=> );(*Level 1 alarm steady*)
tp_almPulse1(IN:=wo_alarmOut.0 , PT:= T#1s, Q=> w_alarmOutp_temp.0, ET=> );(*Level 1 alarm single pulse*)
IF (w_alarmOutp_temp.0 OR wo_alarmOutp.0) AND NOT xi_ack THEN wo_alarmOutp.0:=1; ELSE wo_alarmOutp.0:=0; END_IF(*Level 1 alarm single pulse latched till acknowledge*)

IF ro_perOut < ri_chSP[1] AND NOT(wo_alarmOut.3 OR wo_alarmOut.4)THEN x_alarm2Temp1 := 1; ELSE x_alarm2Temp1 := 0; END_IF
ton_delay2(IN:= x_alarm2Temp1 AND NOT wi_chPara.1 AND NOT wi_chParaJm.1, PT:= REAL_TO_TIME ( ri_chSP[4]*1000), Q=> wo_alarmOut.1, ET=> );(*Level 2 alarm steady*)
tp_almPulse2(IN:=wo_alarmOut.1 , PT:= T#1s, Q=> w_alarmOutp_temp.1, ET=> );(*Level 2 alarm single pulse*)
IF (w_alarmOutp_temp.1 OR wo_alarmOutp.1) AND NOT xi_ack THEN wo_alarmOutp.1:=1; ELSE wo_alarmOutp.1:=0; END_IF(*Level 1 alarm single pulse latched till acknowledge*)

IF ro_perOut > ri_chSP[2]  THEN x_alarm3Temp1 := 1; ELSE x_alarm3Temp1 := 0; END_IF
ton_delay3(IN:= x_alarm3Temp1 AND NOT wi_chPara.2 AND NOT wi_chParaJm.2, PT:= REAL_TO_TIME ( ri_chSP[5]*1000), Q=> wo_alarmOut.2, ET=> );(*Level 3 alarm steady*)
tp_almPulse3(IN:=wo_alarmOut.2 , PT:= T#1s, Q=> w_alarmOutp_temp.2, ET=> );(*Level 3 alarm single pulse*)
IF (w_alarmOutp_temp.2 OR wo_alarmOutp.2) AND NOT xi_ack THEN wo_alarmOutp.2:=1; ELSE wo_alarmOutp.2:=0; END_IF(*Level 1 alarm single pulse latched till acknowledge*)

IF r_sensorValtemp < 3 THEN x_alarm4Temp1 := 1; ELSE x_alarm4Temp1 := 0; END_IF
ton_delay4(IN:= x_alarm4Temp1 AND NOT wi_chPara.3 AND NOT wi_chParaJm.3, PT:= REAL_TO_TIME ( ri_chSP[6]*1000), Q=> wo_alarmOut.3, ET=> );(*cable break alarm steady*)
tp_almPulse4(IN:=wo_alarmOut.3 , PT:= T#1s, Q=> w_alarmOutp_temp.3, ET=> );(*cable break alarm single pulse*)
IF (w_alarmOutp_temp.3 OR wo_alarmOutp.3) AND NOT xi_ack THEN wo_alarmOutp.3:=1; ELSE wo_alarmOutp.3:=0; END_IF(*cable break alarm single pulse latched till acknowledge*)

IF r_sensorValtemp >= 22 THEN x_alarm5Temp1 := 1; ELSE x_alarm5Temp1 := 0; END_IF
ton_delay5(IN:= x_alarm5Temp1 AND NOT wi_chPara.4 AND NOT wi_chParaJm.4, PT:= REAL_TO_TIME ( ri_chSP[6]*1000), Q=> wo_alarmOut.4, ET=> );(*over range alarm steady*)
tp_almPulse5(IN:=wo_alarmOut.4 , PT:= T#1s, Q=> w_alarmOutp_temp.4, ET=> );(*over range alarm single pulse*)
IF (w_alarmOutp_temp.4 OR wo_alarmOutp.4) AND NOT xi_ack THEN wo_alarmOutp.4:=1; ELSE wo_alarmOutp.4:=0; END_IF(*over range alarm single pulse latched till acknowledge*)

IF ro_perOut > ri_chSP[13] THEN x_alarm6Temp1 := 1; ELSE x_alarm6Temp1 := 0; END_IF
ton_delay6(IN:= x_alarm6Temp1 AND NOT wi_chPara.10 AND NOT wi_chParaJm.10, PT:= REAL_TO_TIME ( ri_chSP[14]*1000), Q=> wo_alarmOut.5, ET=> );(*Level 4 alarm steady*)
tp_almPulse6(IN:=wo_alarmOut.5 , PT:= T#1s, Q=> w_alarmOutp_temp.5, ET=> );(*Level 4 alarm single pulse*)
IF (w_alarmOutp_temp.5 OR wo_alarmOutp.5) AND NOT xi_ack THEN wo_alarmOutp.5:=1; ELSE wo_alarmOutp.5:=0; END_IF(*Level 4 alarm single pulse latched till acknowledge*)

(*Alarm message*)
IF	wo_alarmOut.0 AND wo_alarmOut.1 AND NOT wo_alarmOut.3 AND NOT wo_alarmOut.4 AND NOT xi_comErr  THEN	wo_alarmMsg :=1;(*LoLo*)
ELSE IF	NOT wo_alarmOut.0 AND wo_alarmOut.1 AND NOT wo_alarmOut.3 AND NOT wo_alarmOut.4 AND NOT xi_comErr THEN	wo_alarmMsg :=2;(*Lo*)
ELSE IF	NOT wo_alarmOut.5 AND wo_alarmOut.2 AND NOT wo_alarmOut.3 AND NOT wo_alarmOut.4 AND NOT xi_comErr THEN	wo_alarmMsg :=3;(*Hi*)
ELSE IF	wo_alarmOut.5 AND wo_alarmOut.2 AND NOT wo_alarmOut.3 AND NOT wo_alarmOut.4 AND NOT xi_comErr THEN	wo_alarmMsg :=4;(*HiHi*)
ELSE IF	wo_alarmOut.3 OR wo_alarmOut.4 OR xi_comErr THEN	wo_alarmMsg :=5;(*Sensor fault*)
ELSE wo_alarmMsg :=0;	END_IF	END_IF	END_IF	END_IF	END_IF
(*common buzzer out*)
xo_buzPulse := (w_alarmOutp_temp.0 AND NOT wi_chPara.5) OR (w_alarmOutp_temp.1 AND NOT wi_chPara.6) OR (w_alarmOutp_temp.2 AND NOT wi_chPara.7) OR (w_alarmOutp_temp.3 AND NOT wi_chPara.8) OR (w_alarmOutp_temp.4 AND NOT wi_chPara.9) OR (w_alarmOutp_temp.5 AND NOT wi_chPara.11);
(*common indication*)
xo_ind :=wo_alarmOut.0 OR wo_alarmOut.1 OR wo_alarmOut.2 OR wo_alarmOut.3 OR wo_alarmOut.4 OR wo_alarmOut.5;
(*Total inhibited alarms from Jmobile*)
wo_inhTot := BOOL_TO_WORD(wi_chParaJm.0) + BOOL_TO_WORD(wi_chParaJm.1) + BOOL_TO_WORD(wi_chParaJm.2)
 + BOOL_TO_WORD(wi_chParaJm.3) + BOOL_TO_WORD(wi_chParaJm.4) + BOOL_TO_WORD(wi_chParaJm.10);

END_FUNCTION_BLOCK
